KUKA KRL program: f1_Kuka_APT204T03S04.SRC

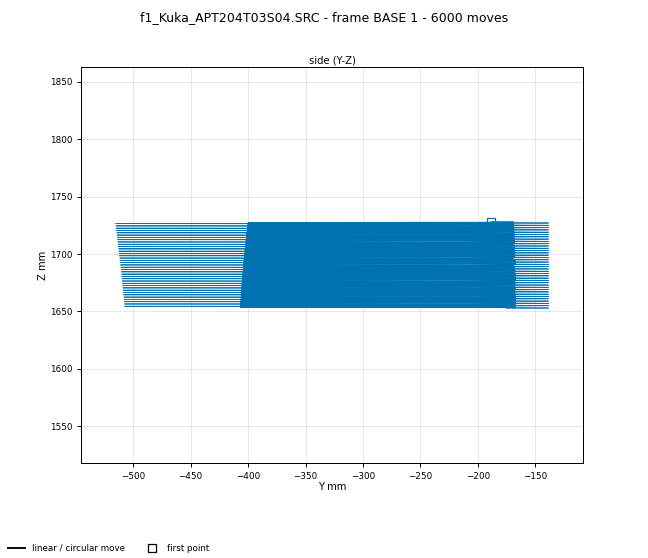
[picture p0: tool path of f1_Kuka_APT204T03S04.SRC in frame BASE 1, 6000 of 6001 moves have a stored position in this frame; points joined in program order, loops and branches not executed]
&ACCESS RVP
&REL 2
&PARAM TEMPLATE = C:\KRC\Roboter\Template\vorgabe
&PARAM EDITMASK = *
DEF f1_Kuka_APT204T03S04()


;FOLD INI;%{PE}%V3.2.0,%MKUKATPBASIS,%CINIT,%VCOMMON,%P
  ;FOLD BAS INI;%{E}%V3.2.0,%MKUKATPBASIS,%CINIT,%VINIT,%P
    GLOBAL INTERRUPT DECL 3 WHEN $STOPMESS==TRUE DO IR_STOPM ( )
    INTERRUPT ON 3
    BAS (#INITMOV,0 )
  ;ENDFOLD (BAS INI)
  ;FOLD USER INI;%{E}%V3.2.0,%MKUKATPUSER,%CINIT,%VINIT,%P
    ;Make your modifications here
  ;ENDFOLD (USER INI)
;ENDFOLD (INI)


;*** Make Null PTP Move
  PTP $pos_act

;*** Auto Load The Correct TOOL Data
  $tool=tool_data[3]

;*** Auto Load The Correct BASE Data
  $base=base_data[1]

  $ADVANCE = 5

;*** Restate Last Velocity
MMPM(30000.0)
SetRPM(6000)
LIN {X 0.021,Y -188.676,Z 1728.125,A 0.000,B 0.000,C 90.000,E1 22.408} C_DIS
LIN {X 0.032,Y -183.742,Z 1728.106,A 0.000,B 0.000,C 90.000,E1 19.087} C_DIS
LIN {X 0.032,Y -179.594,Z 1728.087,A 0.000,B 0.000,C 90.000,E1 15.733} C_DIS
LIN {X 0.087,Y -175.346,Z 1728.064,A 0.000,B 0.000,C 90.000,E1 11.478} C_DIS
LIN {X -0.024,Y -172.220,Z 1728.040,A 0.000,B 0.000,C 90.000,E1 7.239} C_DIS
LIN {X -0.008,Y -169.677,Z 1728.011,A 0.000,B 0.000,C 90.000,E1 2.064} C_DIS
LIN {X 0.036,Y -168.698,Z 1727.969,A 0.000,B 0.000,C 90.000,E1 354.318} C_DIS
LIN {X 0.059,Y -170.485,Z 1727.920,A 0.000,B 0.000,C 90.000,E1 345.644} C_DIS
LIN {X -0.021,Y -173.209,Z 1727.892,A 0.000,B 0.000,C 90.000,E1 340.496} C_DIS
LIN {X -0.074,Y -176.646,Z 1727.868,A 0.000,B 0.000,C 90.000,E1 336.230} C_DIS
LIN {X -0.056,Y -180.954,Z 1727.844,A 0.000,B 0.000,C 90.000,E1 331.975} C_DIS
LIN {X 0.018,Y -185.273,Z 1727.825,A 0.000,B 0.000,C 90.000,E1 328.584} C_DIS
LIN {X -0.017,Y -190.531,Z 1727.807,A 0.000,B 0.000,C 90.000,E1 325.261} C_DIS
LIN {X 0.064,Y -195.194,Z 1727.793,A 0.000,B 0.000,C 90.000,E1 322.763} C_DIS
LIN {X -0.077,Y -200.580,Z 1727.780,A 0.000,B 0.000,C 90.000,E1 320.356} C_DIS
LIN {X 0.012,Y -207.729,Z 1727.764,A 0.000,B 0.000,C 90.000,E1 317.514} C_DIS
LIN {X -0.032,Y -215.873,Z 1727.749,A 0.000,B 0.000,C 90.000,E1 314.757} C_DIS
LIN {X 0.037,Y -223.797,Z 1727.736,A 0.000,B 0.000,C 90.000,E1 312.405} C_DIS
LIN {X 0.016,Y -231.179,Z 1727.725,A 0.000,B 0.000,C 90.000,E1 310.496} C_DIS
LIN {X -0.046,Y -239.468,Z 1727.714,A 0.000,B 0.000,C 90.000,E1 308.624} C_DIS
LIN {X 0.070,Y -248.697,Z 1727.704,A 0.000,B 0.000,C 90.000,E1 306.744} C_DIS
LIN {X -0.140,Y -261.217,Z 1727.692,A 0.000,B 0.000,C 90.000,E1 304.612} C_DIS
LIN {X 0.044,Y -279.547,Z 1727.676,A 0.000,B 0.000,C 90.000,E1 301.750} C_DIS
LIN {X 0.044,Y -301.889,Z 1727.659,A 0.000,B 0.000,C 90.000,E1 298.693} C_DIS
LIN {X -0.011,Y -320.034,Z 1727.647,A 0.000,B 0.000,C 90.000,E1 296.411} C_DIS
LIN {X -0.057,Y -335.844,Z 1727.636,A 0.000,B 0.000,C 90.000,E1 294.515} C_DIS
LIN {X 0.099,Y -348.845,Z 1727.628,A 0.000,B 0.000,C 90.000,E1 292.950} C_DIS
LIN {X -0.069,Y -361.378,Z 1727.619,A 0.000,B 0.000,C 90.000,E1 291.461} C_DIS
LIN {X 0.072,Y -371.097,Z 1727.613,A 0.000,B 0.000,C 90.000,E1 290.248} C_DIS
LIN {X -0.125,Y -377.905,Z 1727.608,A 0.000,B 0.000,C 90.000,E1 289.396} C_DIS
LIN {X 0.102,Y -381.961,Z 1727.604,A 0.000,B 0.000,C 90.000,E1 288.779} C_DIS
LIN {X -0.113,Y -387.245,Z 1727.600,A 0.000,B 0.000,C 90.000,E1 287.946} C_DIS
LIN {X 0.057,Y -390.219,Z 1727.596,A 0.000,B 0.000,C 90.000,E1 287.347} C_DIS
LIN {X 0.030,Y -393.882,Z 1727.592,A 0.000,B 0.000,C 90.000,E1 286.496} C_DIS
LIN {X -0.134,Y -395.829,Z 1727.589,A 0.000,B 0.000,C 90.000,E1 285.953} C_DIS
LIN {X -0.018,Y -397.436,Z 1727.585,A 0.000,B 0.000,C 90.000,E1 285.371} C_DIS
LIN {X -0.169,Y -398.668,Z 1727.582,A 0.000,B 0.000,C 90.000,E1 284.828} C_DIS
LIN {X -0.025,Y -399.563,Z 1727.579,A 0.000,B 0.000,C 90.000,E1 284.245} C_DIS
LIN {X 0.225,Y -400.068,Z 1727.576,A 0.000,B 0.000,C 90.000,E1 283.647} C_DIS
LIN {X -0.004,Y -400.218,Z 1727.573,A 0.000,B 0.000,C 90.000,E1 283.119} C_DIS
LIN {X 0.160,Y -399.926,Z 1727.570,A 0.000,B 0.000,C 90.000,E1 282.535} C_DIS
LIN {X -0.063,Y -399.279,Z 1727.567,A 0.000,B 0.000,C 90.000,E1 282.007} C_DIS
LIN {X 0.103,Y -398.089,Z 1727.564,A 0.000,B 0.000,C 90.000,E1 281.422} C_DIS
LIN {X -0.126,Y -396.417,Z 1727.560,A 0.000,B 0.000,C 90.000,E1 280.894} C_DIS
LIN {X 0.026,Y -394.202,Z 1727.557,A 0.000,B 0.000,C 90.000,E1 280.310} C_DIS
LIN {X 0.159,Y -391.354,Z 1727.554,A 0.000,B 0.000,C 90.000,E1 279.726} C_DIS
LIN {X -0.031,Y -379.747,Z 1727.543,A 0.000,B 0.000,C 90.000,E1 277.757} C_DIS
LIN {X -0.040,Y -376.170,Z 1727.540,A 0.000,B 0.000,C 90.000,E1 277.182} C_DIS
LIN {X -0.068,Y -372.156,Z 1727.537,A 0.000,B 0.000,C 90.000,E1 276.606} C_DIS
LIN {X -0.115,Y -367.505,Z 1727.533,A 0.000,B 0.000,C 90.000,E1 276.030} C_DIS
LIN {X -0.141,Y -362.126,Z 1727.530,A 0.000,B 0.000,C 90.000,E1 275.448} C_DIS
LIN {X -0.100,Y -356.268,Z 1727.527,A 0.000,B 0.000,C 90.000,E1 274.878} C_DIS
LIN {X -0.130,Y -350.292,Z 1727.524,A 0.000,B 0.000,C 90.000,E1 274.359} C_DIS
LIN {X 0.065,Y -344.121,Z 1727.521,A 0.000,B 0.000,C 90.000,E1 273.841} C_DIS
LIN {X 0.135,Y -337.795,Z 1727.519,A 0.000,B 0.000,C 90.000,E1 273.383} C_DIS
LIN {X 0.110,Y -331.427,Z 1727.517,A 0.000,B 0.000,C 90.000,E1 272.980} C_DIS
LIN {X -0.017,Y -321.523,Z 1727.514,A 0.000,B 0.000,C 90.000,E1 272.465} C_DIS
LIN {X -0.159,Y -314.709,Z 1727.512,A 0.000,B 0.000,C 90.000,E1 272.178} C_DIS
LIN {X -0.109,Y -307.490,Z 1727.510,A 0.000,B 0.000,C 90.000,E1 271.892} C_DIS
LIN {X -0.010,Y -296.875,Z 1727.509,A 0.000,B 0.000,C 90.000,E1 271.547} C_DIS
LIN {X -0.063,Y -289.643,Z 1727.508,A 0.000,B 0.000,C 90.000,E1 271.375} C_DIS
LIN {X -0.035,Y -277.079,Z 1727.506,A 0.000,B 0.000,C 90.000,E1 271.146} C_DIS
LIN {X -0.052,Y -264.431,Z 1727.505,A 0.000,B 0.000,C 90.000,E1 270.974} C_DIS
LIN {X -0.027,Y -253.912,Z 1727.505,A 0.000,B 0.000,C 90.000,E1 270.859} C_DIS
LIN {X -0.046,Y -239.564,Z 1727.504,A 0.000,B 0.000,C 90.000,E1 270.802} C_DIS
LIN {X -0.067,Y -181.507,Z 1727.504,A 0.000,B 0.000,C 90.000,E1 270.802} C_DIS
LIN {X -0.020,Y -181.537,Z 1727.499,A 0.000,B 0.000,C 90.000,E1 269.885} C_DIS
LIN {X -0.036,Y -180.813,Z 1727.471,A 0.000,B 0.000,C 90.000,E1 264.837} C_DIS
LIN {X 0.041,Y -178.916,Z 1727.443,A 0.000,B 0.000,C 90.000,E1 259.746} C_DIS
LIN {X -0.050,Y -175.961,Z 1727.415,A 0.000,B 0.000,C 90.000,E1 254.685} C_DIS
LIN {X 0.067,Y -175.435,Z 1727.410,A 0.000,B 0.000,C 90.000,E1 253.795} C_DIS
LIN {X 0.069,Y -172.193,Z 1727.386,A 0.000,B 0.000,C 90.000,E1 249.518} C_DIS
LIN {X 0.046,Y -171.666,Z 1727.382,A 0.000,B 0.000,C 90.000,E1 248.666} C_DIS
LIN {X 0.029,Y -167.891,Z 1727.358,A 0.000,B 0.000,C 90.000,E1 244.357} C_DIS
LIN {X 0.045,Y -166.629,Z 1727.348,A 0.000,B 0.000,C 90.000,E1 242.615} C_DIS
LIN {X 0.037,Y -162.615,Z 1727.324,A 0.000,B 0.000,C 90.000,E1 238.250} C_DIS
LIN {X 0.012,Y -161.301,Z 1727.314,A 0.000,B 0.000,C 90.000,E1 236.501} C_DIS
LIN {X 0.045,Y -157.299,Z 1727.289,A 0.000,B 0.000,C 90.000,E1 232.065} C_DIS
LIN {X 0.074,Y -155.274,Z 1727.275,A 0.000,B 0.000,C 90.000,E1 229.380} C_DIS
LIN {X 0.002,Y -151.641,Z 1727.250,A 0.000,B 0.000,C 90.000,E1 224.919} C_DIS
LIN {X 0.049,Y -150.509,Z 1727.240,A 0.000,B 0.000,C 90.000,E1 223.095} C_DIS
LIN {X -0.037,Y -147.234,Z 1727.214,A 0.000,B 0.000,C 90.000,E1 218.588} C_DIS
LIN {X 0.048,Y -145.257,Z 1727.194,A 0.000,B 0.000,C 90.000,E1 214.898} C_DIS
LIN {X -0.036,Y -142.370,Z 1727.163,A 0.000,B 0.000,C 90.000,E1 209.411} C_DIS
LIN {X 0.085,Y -141.755,Z 1727.153,A 0.000,B 0.000,C 90.000,E1 207.513} C_DIS
LIN {X 0.010,Y -139.497,Z 1727.117,A 0.000,B 0.000,C 90.000,E1 201.046} C_DIS
LIN {X 0.047,Y -139.002,Z 1727.101,A 0.000,B 0.000,C 90.000,E1 198.236} C_DIS
LIN {X 0.003,Y -138.338,Z 1727.055,A 0.000,B 0.000,C 90.000,E1 189.849} C_DIS
LIN {X 0.025,Y -139.408,Z 1727.008,A 0.000,B 0.000,C 90.000,E1 181.432} C_DIS
LIN {X -0.062,Y -141.318,Z 1726.972,A 0.000,B 0.000,C 90.000,E1 174.951} C_DIS
LIN {X 0.037,Y -142.677,Z 1726.956,A 0.000,B 0.000,C 90.000,E1 172.129} C_DIS
LIN {X 0.017,Y -145.032,Z 1726.931,A 0.000,B 0.000,C 90.000,E1 167.521} C_DIS
LIN {X -0.026,Y -147.657,Z 1726.910,A 0.000,B 0.000,C 90.000,E1 163.866} C_DIS
LIN {X 0.050,Y -150.295,Z 1726.890,A 0.000,B 0.000,C 90.000,E1 160.188} C_DIS
LIN {X -0.079,Y -153.704,Z 1726.870,A 0.000,B 0.000,C 90.000,E1 156.613} C_DIS
LIN {X -0.024,Y -157.118,Z 1726.850,A 0.000,B 0.000,C 90.000,E1 152.999} C_DIS
LIN {X 0.052,Y -161.260,Z 1726.830,A 0.000,B 0.000,C 90.000,E1 149.410} C_DIS
LIN {X -0.020,Y -164.379,Z 1726.815,A 0.000,B 0.000,C 90.000,E1 146.786} C_DIS
LIN {X -0.033,Y -169.054,Z 1726.796,A 0.000,B 0.000,C 90.000,E1 143.290} C_DIS
LIN {X 0.019,Y -171.615,Z 1726.786,A 0.000,B 0.000,C 90.000,E1 141.537} C_DIS
LIN {X 0.067,Y -176.571,Z 1726.767,A 0.000,B 0.000,C 90.000,E1 138.081} C_DIS
LIN {X -0.060,Y -180.869,Z 1726.753,A 0.000,B 0.000,C 90.000,E1 135.567} C_DIS
LIN {X 0.062,Y -186.283,Z 1726.734,A 0.000,B 0.000,C 90.000,E1 132.162} C_DIS
LIN {X -0.017,Y -190.918,Z 1726.720,A 0.000,B 0.000,C 90.000,E1 129.688} C_DIS
LIN {X 0.051,Y -196.685,Z 1726.702,A 0.000,B 0.000,C 90.000,E1 126.377} C_DIS
LIN {X 0.081,Y -199.929,Z 1726.693,A 0.000,B 0.000,C 90.000,E1 124.739} C_DIS
LIN {X -0.026,Y -205.846,Z 1726.675,A 0.000,B 0.000,C 90.000,E1 121.544} C_DIS
LIN {X -0.035,Y -209.790,Z 1726.664,A 0.000,B 0.000,C 90.000,E1 119.617} C_DIS
LIN {X -0.091,Y -333.994,Z 1726.664,A 0.000,B 0.000,C 90.000,E1 119.617} C_DIS
LIN {X -0.010,Y -338.536,Z 1726.664,A 0.000,B 0.000,C 90.000,E1 119.489} C_DIS
LIN {X 0.072,Y -340.616,Z 1726.663,A 0.000,B 0.000,C 90.000,E1 119.361} C_DIS
LIN {X -0.059,Y -343.462,Z 1726.662,A 0.000,B 0.000,C 90.000,E1 119.155} C_DIS
LIN {X -0.065,Y -347.189,Z 1726.659,A 0.000,B 0.000,C 90.000,E1 118.693} C_DIS
LIN {X 0.099,Y -348.907,Z 1726.658,A 0.000,B 0.000,C 90.000,E1 118.359} C_DIS
LIN {X -0.093,Y -361.834,Z 1726.643,A 0.000,B 0.000,C 90.000,E1 115.668} C_DIS
LIN {X -0.076,Y -376.245,Z 1726.628,A 0.000,B 0.000,C 90.000,E1 113.003} C_DIS
LIN {X 0.097,Y -390.434,Z 1726.615,A 0.000,B 0.000,C 90.000,E1 110.663} C_DIS
LIN {X -0.010,Y -406.020,Z 1726.602,A 0.000,B 0.000,C 90.000,E1 108.417} C_DIS
LIN {X 0.018,Y -423.110,Z 1726.590,A 0.000,B 0.000,C 90.000,E1 106.205} C_DIS
LIN {X -0.058,Y -441.822,Z 1726.578,A 0.000,B 0.000,C 90.000,E1 104.064} C_DIS
LIN {X 0.100,Y -461.716,Z 1726.567,A 0.000,B 0.000,C 90.000,E1 102.007} C_DIS
LIN {X 0.139,Y -484.774,Z 1726.555,A 0.000,B 0.000,C 90.000,E1 99.905} C_DIS
LIN {X 0.179,Y -508.285,Z 1726.545,A 0.000,B 0.000,C 90.000,E1 97.992} C_DIS
LIN {X -0.039,Y -510.226,Z 1726.543,A 0.000,B 0.000,C 90.000,E1 97.814} C_DIS
LIN {X -0.158,Y -511.971,Z 1726.542,A 0.000,B 0.000,C 90.000,E1 97.587} C_DIS
LIN {X -0.211,Y -513.277,Z 1726.541,A 0.000,B 0.000,C 90.000,E1 97.352} C_DIS
LIN {X 0.150,Y -514.880,Z 1726.538,A 0.000,B 0.000,C 90.000,E1 96.834} C_DIS
LIN {X 0.006,Y -515.381,Z 1726.535,A 0.000,B 0.000,C 90.000,E1 96.372} C_DIS
LIN {X -0.129,Y -514.864,Z 1726.533,A 0.000,B 0.000,C 90.000,E1 95.910} C_DIS
LIN {X 0.249,Y -513.239,Z 1726.530,A 0.000,B 0.000,C 90.000,E1 95.391} C_DIS
LIN {X 0.157,Y -511.916,Z 1726.529,A 0.000,B 0.000,C 90.000,E1 95.163} C_DIS
LIN {X 0.131,Y -501.107,Z 1726.521,A 0.000,B 0.000,C 90.000,E1 93.726} C_DIS
LIN {X -0.234,Y -488.498,Z 1726.511,A 0.000,B 0.000,C 90.000,E1 92.064} C_DIS
LIN {X 0.126,Y -475.702,Z 1726.502,A 0.000,B 0.000,C 90.000,E1 90.286} C_DIS
LIN {X -0.052,Y -464.718,Z 1726.493,A 0.000,B 0.000,C 90.000,E1 88.797} C_DIS
LIN {X -0.170,Y -451.882,Z 1726.483,A 0.000,B 0.000,C 90.000,E1 87.020} C_DIS
LIN {X 0.127,Y -437.184,Z 1726.472,A 0.000,B 0.000,C 90.000,E1 84.894} C_DIS
LIN {X -0.047,Y -424.340,Z 1726.461,A 0.000,B 0.000,C 90.000,E1 83.053} C_DIS
LIN {X -0.059,Y -406.525,Z 1726.446,A 0.000,B 0.000,C 90.000,E1 80.330} C_DIS
LIN {X 0.031,Y -389.797,Z 1726.431,A 0.000,B 0.000,C 90.000,E1 77.521} C_DIS
LIN {X 0.060,Y -377.038,Z 1726.418,A 0.000,B 0.000,C 90.000,E1 75.227} C_DIS
LIN {X -0.004,Y -366.137,Z 1726.407,A 0.000,B 0.000,C 90.000,E1 73.196} C_DIS
LIN {X 0.137,Y -352.444,Z 1726.392,A 0.000,B 0.000,C 90.000,E1 70.496} C_DIS
LIN {X -0.072,Y -339.450,Z 1726.377,A 0.000,B 0.000,C 90.000,E1 67.794} C_DIS
LIN {X -0.006,Y -329.467,Z 1726.365,A 0.000,B 0.000,C 90.000,E1 65.613} C_DIS
LIN {X 0.136,Y -317.003,Z 1726.349,A 0.000,B 0.000,C 90.000,E1 62.743} C_DIS
LIN {X 0.005,Y -307.384,Z 1726.336,A 0.000,B 0.000,C 90.000,E1 60.511} C_DIS
LIN {X 0.090,Y -297.798,Z 1726.323,A 0.000,B 0.000,C 90.000,E1 58.201} C_DIS
LIN {X 0.015,Y -288.121,Z 1726.310,A 0.000,B 0.000,C 90.000,E1 55.881} C_DIS
LIN {X 0.057,Y -278.348,Z 1726.297,A 0.000,B 0.000,C 90.000,E1 53.497} C_DIS
LIN {X -0.007,Y -268.542,Z 1726.284,A 0.000,B 0.000,C 90.000,E1 51.090} C_DIS
LIN {X 0.107,Y -257.502,Z 1726.268,A 0.000,B 0.000,C 90.000,E1 48.243} C_DIS
LIN {X 0.086,Y -245.401,Z 1726.250,A 0.000,B 0.000,C 90.000,E1 45.000} C_DIS
LIN {X 0.076,Y -234.032,Z 1726.232,A 0.000,B 0.000,C 90.000,E1 41.676} C_DIS
LIN {X 0.026,Y -224.586,Z 1726.215,A 0.000,B 0.000,C 90.000,E1 38.669} C_DIS
LIN {X -0.089,Y -217.046,Z 1726.200,A 0.000,B 0.000,C 90.000,E1 36.011} C_DIS
LIN {X -0.046,Y -209.230,Z 1726.183,A 0.000,B 0.000,C 90.000,E1 32.880} C_DIS
LIN {X 0.102,Y -202.113,Z 1726.165,A 0.000,B 0.000,C 90.000,E1 29.667} C_DIS
LIN {X -0.046,Y -195.705,Z 1726.147,A 0.000,B 0.000,C 90.000,E1 26.488} C_DIS
LIN {X 0.008,Y -189.907,Z 1726.129,A 0.000,B 0.000,C 90.000,E1 23.206} C_DIS
LIN {X -0.020,Y -185.956,Z 1726.115,A 0.000,B 0.000,C 90.000,E1 20.737} C_DIS
LIN {X -0.027,Y -181.437,Z 1726.097,A 0.000,B 0.000,C 90.000,E1 17.402} C_DIS
LIN {X -0.002,Y -176.803,Z 1726.073,A 0.000,B 0.000,C 90.000,E1 13.175} C_DIS
LIN {X -0.012,Y -173.238,Z 1726.050,A 0.000,B 0.000,C 90.000,E1 8.916} C_DIS
LIN {X 0.080,Y -170.204,Z 1726.021,A 0.000,B 0.000,C 90.000,E1 3.726} C_DIS
LIN {X 0.031,Y -168.549,Z 1725.969,A 0.000,B 0.000,C 90.000,E1 354.318} C_DIS
LIN {X 0.047,Y -170.375,Z 1725.920,A 0.000,B 0.000,C 90.000,E1 345.644} C_DIS
LIN {X -0.036,Y -173.138,Z 1725.892,A 0.000,B 0.000,C 90.000,E1 340.496} C_DIS
LIN {X 0.069,Y -176.589,Z 1725.868,A 0.000,B 0.000,C 90.000,E1 336.177} C_DIS
LIN {X -0.077,Y -180.926,Z 1725.844,A 0.000,B 0.000,C 90.000,E1 331.975} C_DIS
LIN {X -0.004,Y -185.262,Z 1725.825,A 0.000,B 0.000,C 90.000,E1 328.584} C_DIS
LIN {X -0.040,Y -190.547,Z 1725.807,A 0.000,B 0.000,C 90.000,E1 325.261} C_DIS
LIN {X 0.041,Y -195.244,Z 1725.793,A 0.000,B 0.000,C 90.000,E1 322.763} C_DIS
LIN {X 0.050,Y -201.625,Z 1725.777,A 0.000,B 0.000,C 90.000,E1 319.908} C_DIS
LIN {X 0.031,Y -208.936,Z 1725.762,A 0.000,B 0.000,C 90.000,E1 317.106} C_DIS
LIN {X 0.008,Y -217.290,Z 1725.746,A 0.000,B 0.000,C 90.000,E1 314.352} C_DIS
LIN {X 0.105,Y -225.385,Z 1725.734,A 0.000,B 0.000,C 90.000,E1 312.000} C_DIS
LIN {X 0.104,Y -232.950,Z 1725.723,A 0.000,B 0.000,C 90.000,E1 310.092} C_DIS
LIN {X -0.076,Y -241.392,Z 1725.712,A 0.000,B 0.000,C 90.000,E1 308.257} C_DIS
LIN {X 0.065,Y -250.866,Z 1725.702,A 0.000,B 0.000,C 90.000,E1 306.377} C_DIS
LIN {X 0.109,Y -263.640,Z 1725.690,A 0.000,B 0.000,C 90.000,E1 304.199} C_DIS
LIN {X -0.011,Y -282.177,Z 1725.675,A 0.000,B 0.000,C 90.000,E1 301.416} C_DIS
LIN {X 0.056,Y -302.095,Z 1725.659,A 0.000,B 0.000,C 90.000,E1 298.693} C_DIS
LIN {X 0.005,Y -320.201,Z 1725.647,A 0.000,B 0.000,C 90.000,E1 296.411} C_DIS
LIN {X -0.055,Y -335.995,Z 1725.636,A 0.000,B 0.000,C 90.000,E1 294.515} C_DIS
LIN {X 0.102,Y -348.973,Z 1725.628,A 0.000,B 0.000,C 90.000,E1 292.950} C_DIS
LIN {X -0.065,Y -361.513,Z 1725.619,A 0.000,B 0.000,C 90.000,E1 291.461} C_DIS
LIN {X 0.078,Y -371.239,Z 1725.613,A 0.000,B 0.000,C 90.000,E1 290.248} C_DIS
LIN {X -0.117,Y -378.062,Z 1725.608,A 0.000,B 0.000,C 90.000,E1 289.396} C_DIS
LIN {X 0.112,Y -382.108,Z 1725.604,A 0.000,B 0.000,C 90.000,E1 288.779} C_DIS
LIN {X -0.103,Y -387.404,Z 1725.600,A 0.000,B 0.000,C 90.000,E1 287.946} C_DIS
LIN {X 0.068,Y -390.382,Z 1725.596,A 0.000,B 0.000,C 90.000,E1 287.347} C_DIS
LIN {X 0.043,Y -394.065,Z 1725.592,A 0.000,B 0.000,C 90.000,E1 286.496} C_DIS
LIN {X -0.120,Y -396.048,Z 1725.589,A 0.000,B 0.000,C 90.000,E1 285.953} C_DIS
LIN {X -0.003,Y -397.675,Z 1725.585,A 0.000,B 0.000,C 90.000,E1 285.371} C_DIS
LIN {X -0.152,Y -398.895,Z 1725.582,A 0.000,B 0.000,C 90.000,E1 284.828} C_DIS
LIN {X -0.007,Y -399.799,Z 1725.579,A 0.000,B 0.000,C 90.000,E1 284.245} C_DIS
LIN {X -0.144,Y -400.296,Z 1725.576,A 0.000,B 0.000,C 90.000,E1 283.703} C_DIS
LIN {X 0.017,Y -400.428,Z 1725.573,A 0.000,B 0.000,C 90.000,E1 283.119} C_DIS
LIN {X 0.183,Y -400.155,Z 1725.570,A 0.000,B 0.000,C 90.000,E1 282.535} C_DIS
LIN {X -0.040,Y -399.488,Z 1725.567,A 0.000,B 0.000,C 90.000,E1 282.007} C_DIS
LIN {X 0.128,Y -398.290,Z 1725.564,A 0.000,B 0.000,C 90.000,E1 281.422} C_DIS
LIN {X -0.100,Y -396.610,Z 1725.560,A 0.000,B 0.000,C 90.000,E1 280.894} C_DIS
LIN {X 0.052,Y -394.381,Z 1725.557,A 0.000,B 0.000,C 90.000,E1 280.310} C_DIS
LIN {X 0.186,Y -391.546,Z 1725.554,A 0.000,B 0.000,C 90.000,E1 279.726} C_DIS
LIN {X 0.000,Y -379.916,Z 1725.543,A 0.000,B 0.000,C 90.000,E1 277.757} C_DIS
LIN {X 0.006,Y -374.386,Z 1725.538,A 0.000,B 0.000,C 90.000,E1 276.891} C_DIS
LIN {X -0.033,Y -370.048,Z 1725.535,A 0.000,B 0.000,C 90.000,E1 276.315} C_DIS
LIN {X -0.093,Y -364.999,Z 1725.532,A 0.000,B 0.000,C 90.000,E1 275.739} C_DIS
LIN {X 0.179,Y -359.290,Z 1725.529,A 0.000,B 0.000,C 90.000,E1 275.106} C_DIS
LIN {X 0.013,Y -353.325,Z 1725.526,A 0.000,B 0.000,C 90.000,E1 274.588} C_DIS
LIN {X 0.089,Y -347.232,Z 1725.523,A 0.000,B 0.000,C 90.000,E1 274.073} C_DIS
LIN {X 0.076,Y -340.957,Z 1725.520,A 0.000,B 0.000,C 90.000,E1 273.612} C_DIS
LIN {X -0.061,Y -334.532,Z 1725.518,A 0.000,B 0.000,C 90.000,E1 273.212} C_DIS
LIN {X 0.026,Y -327.904,Z 1725.516,A 0.000,B 0.000,C 90.000,E1 272.808} C_DIS
LIN {X 0.012,Y -321.289,Z 1725.514,A 0.000,B 0.000,C 90.000,E1 272.465} C_DIS
LIN {X -0.146,Y -314.295,Z 1725.512,A 0.000,B 0.000,C 90.000,E1 272.178} C_DIS
LIN {X -0.009,Y -303.873,Z 1725.510,A 0.000,B 0.000,C 90.000,E1 271.776} C_DIS
LIN {X -0.087,Y -293.320,Z 1725.508,A 0.000,B 0.000,C 90.000,E1 271.489} C_DIS
LIN {X -0.080,Y -285.623,Z 1725.507,A 0.000,B 0.000,C 90.000,E1 271.318} C_DIS
LIN {X 0.077,Y -269.385,Z 1725.506,A 0.000,B 0.000,C 90.000,E1 271.031} C_DIS
LIN {X 0.089,Y -255.161,Z 1725.505,A 0.000,B 0.000,C 90.000,E1 270.859} C_DIS
LIN {X 0.059,Y -239.893,Z 1725.505,A 0.000,B 0.000,C 90.000,E1 270.802} C_DIS
LIN {X 0.014,Y -181.500,Z 1725.505,A 0.000,B 0.000,C 90.000,E1 270.802} C_DIS
LIN {X 0.068,Y -181.543,Z 1725.500,A 0.000,B 0.000,C 90.000,E1 269.885} C_DIS
LIN {X 0.052,Y -180.822,Z 1725.471,A 0.000,B 0.000,C 90.000,E1 264.837} C_DIS
LIN {X -0.048,Y -178.926,Z 1725.443,A 0.000,B 0.000,C 90.000,E1 259.803} C_DIS
LIN {X -0.010,Y -175.973,Z 1725.415,A 0.000,B 0.000,C 90.000,E1 254.700} C_DIS
LIN {X -0.065,Y -175.459,Z 1725.410,A 0.000,B 0.000,C 90.000,E1 253.866} C_DIS
LIN {X -0.007,Y -172.210,Z 1725.386,A 0.000,B 0.000,C 90.000,E1 249.571} C_DIS
LIN {X -0.029,Y -171.686,Z 1725.382,A 0.000,B 0.000,C 90.000,E1 248.720} C_DIS
LIN {X -0.039,Y -167.912,Z 1725.358,A 0.000,B 0.000,C 90.000,E1 244.409} C_DIS
LIN {X -0.020,Y -166.654,Z 1725.348,A 0.000,B 0.000,C 90.000,E1 242.666} C_DIS
LIN {X 0.034,Y -162.638,Z 1725.324,A 0.000,B 0.000,C 90.000,E1 238.280} C_DIS
LIN {X -0.041,Y -161.325,Z 1725.314,A 0.000,B 0.000,C 90.000,E1 236.548} C_DIS
LIN {X 0.002,Y -157.321,Z 1725.290,A 0.000,B 0.000,C 90.000,E1 232.110} C_DIS
LIN {X -0.065,Y -155.301,Z 1725.275,A 0.000,B 0.000,C 90.000,E1 229.461} C_DIS
LIN {X 0.081,Y -151.661,Z 1725.250,A 0.000,B 0.000,C 90.000,E1 224.919} C_DIS
LIN {X 0.018,Y -150.527,Z 1725.240,A 0.000,B 0.000,C 90.000,E1 223.137} C_DIS
LIN {X -0.051,Y -147.252,Z 1725.214,A 0.000,B 0.000,C 90.000,E1 218.624} C_DIS
LIN {X 0.005,Y -145.277,Z 1725.194,A 0.000,B 0.000,C 90.000,E1 214.945} C_DIS
LIN {X 0.039,Y -142.381,Z 1725.163,A 0.000,B 0.000,C 90.000,E1 209.411} C_DIS
LIN {X -0.039,Y -141.359,Z 1725.148,A 0.000,B 0.000,C 90.000,E1 206.668} C_DIS
LIN {X 0.071,Y -139.342,Z 1725.112,A 0.000,B 0.000,C 90.000,E1 200.120} C_DIS
LIN {X -0.011,Y -139.010,Z 1725.102,A 0.000,B 0.000,C 90.000,E1 198.290} C_DIS
LIN {X -0.059,Y -138.341,Z 1725.055,A 0.000,B 0.000,C 90.000,E1 189.905} C_DIS
LIN {X -0.039,Y -139.400,Z 1725.008,A 0.000,B 0.000,C 90.000,E1 181.489} C_DIS
LIN {X 0.014,Y -141.304,Z 1724.972,A 0.000,B 0.000,C 90.000,E1 174.951} C_DIS
LIN {X -0.028,Y -142.665,Z 1724.957,A 0.000,B 0.000,C 90.000,E1 172.186} C_DIS
LIN {X -0.079,Y -145.012,Z 1724.931,A 0.000,B 0.000,C 90.000,E1 167.589} C_DIS
LIN {X 0.052,Y -147.639,Z 1724.911,A 0.000,B 0.000,C 90.000,E1 163.866} C_DIS
LIN {X -0.012,Y -150.271,Z 1724.890,A 0.000,B 0.000,C 90.000,E1 160.242} C_DIS
LIN {X 0.001,Y -153.672,Z 1724.870,A 0.000,B 0.000,C 90.000,E1 156.613} C_DIS
LIN {X 0.057,Y -157.087,Z 1724.850,A 0.000,B 0.000,C 90.000,E1 152.999} C_DIS
LIN {X -0.004,Y -161.222,Z 1724.830,A 0.000,B 0.000,C 90.000,E1 149.459} C_DIS
LIN {X 0.080,Y -163.312,Z 1724.820,A 0.000,B 0.000,C 90.000,E1 147.661} C_DIS
LIN {X -0.048,Y -167.761,Z 1724.801,A 0.000,B 0.000,C 90.000,E1 144.196} C_DIS
LIN {X 0.104,Y -171.578,Z 1724.786,A 0.000,B 0.000,C 90.000,E1 141.537} C_DIS
LIN {X -0.096,Y -176.527,Z 1724.767,A 0.000,B 0.000,C 90.000,E1 138.162} C_DIS
LIN {X 0.028,Y -180.825,Z 1724.753,A 0.000,B 0.000,C 90.000,E1 135.567} C_DIS
LIN {X 0.013,Y -186.235,Z 1724.734,A 0.000,B 0.000,C 90.000,E1 132.204} C_DIS
LIN {X -0.048,Y -190.871,Z 1724.721,A 0.000,B 0.000,C 90.000,E1 129.725} C_DIS
LIN {X -0.015,Y -196.634,Z 1724.702,A 0.000,B 0.000,C 90.000,E1 126.423} C_DIS
LIN {X -0.103,Y -199.873,Z 1724.693,A 0.000,B 0.000,C 90.000,E1 124.818} C_DIS
LIN {X 0.093,Y -204.269,Z 1724.680,A 0.000,B 0.000,C 90.000,E1 122.339} C_DIS
LIN {X 0.061,Y -209.734,Z 1724.665,A 0.000,B 0.000,C 90.000,E1 119.617} C_DIS
LIN {X 0.061,Y -334.184,Z 1724.665,A 0.000,B 0.000,C 90.000,E1 119.617} C_DIS
LIN {X -0.151,Y -338.440,Z 1724.664,A 0.000,B 0.000,C 90.000,E1 119.539} C_DIS
LIN {X -0.069,Y -340.506,Z 1724.663,A 0.000,B 0.000,C 90.000,E1 119.411} C_DIS
LIN {X 0.097,Y -343.339,Z 1724.662,A 0.000,B 0.000,C 90.000,E1 119.155} C_DIS
LIN {X 0.084,Y -347.067,Z 1724.659,A 0.000,B 0.000,C 90.000,E1 118.693} C_DIS
LIN {X -0.058,Y -348.777,Z 1724.658,A 0.000,B 0.000,C 90.000,E1 118.409} C_DIS
LIN {X 0.058,Y -361.691,Z 1724.643,A 0.000,B 0.000,C 90.000,E1 115.668} C_DIS
LIN {X -0.070,Y -376.087,Z 1724.628,A 0.000,B 0.000,C 90.000,E1 113.025} C_DIS
LIN {X 0.113,Y -390.262,Z 1724.615,A 0.000,B 0.000,C 90.000,E1 110.684} C_DIS
LIN {X 0.147,Y -405.833,Z 1724.602,A 0.000,B 0.000,C 90.000,E1 108.417} C_DIS
LIN {X 0.176,Y -422.907,Z 1724.590,A 0.000,B 0.000,C 90.000,E1 106.205} C_DIS
LIN {X 0.102,Y -441.603,Z 1724.578,A 0.000,B 0.000,C 90.000,E1 104.064} C_DIS
LIN {X -0.197,Y -461.489,Z 1724.567,A 0.000,B 0.000,C 90.000,E1 102.063} C_DIS
LIN {X -0.192,Y -484.541,Z 1724.555,A 0.000,B 0.000,C 90.000,E1 99.962} C_DIS
LIN {X -0.185,Y -508.048,Z 1724.545,A 0.000,B 0.000,C 90.000,E1 98.049} C_DIS
LIN {X 0.099,Y -509.989,Z 1724.543,A 0.000,B 0.000,C 90.000,E1 97.814} C_DIS
LIN {X -0.020,Y -511.734,Z 1724.542,A 0.000,B 0.000,C 90.000,E1 97.587} C_DIS
LIN {X -0.072,Y -513.038,Z 1724.541,A 0.000,B 0.000,C 90.000,E1 97.352} C_DIS
LIN {X -0.224,Y -514.635,Z 1724.538,A 0.000,B 0.000,C 90.000,E1 96.891} C_DIS
LIN {X 0.142,Y -515.135,Z 1724.536,A 0.000,B 0.000,C 90.000,E1 96.372} C_DIS
LIN {X 0.005,Y -514.617,Z 1724.533,A 0.000,B 0.000,C 90.000,E1 95.910} C_DIS
LIN {X -0.129,Y -512.990,Z 1724.530,A 0.000,B 0.000,C 90.000,E1 95.448} C_DIS
LIN {X -0.221,Y -511.668,Z 1724.529,A 0.000,B 0.000,C 90.000,E1 95.220} C_DIS
LIN {X -0.130,Y -502.681,Z 1724.522,A 0.000,B 0.000,C 90.000,E1 94.012} C_DIS
LIN {X 0.020,Y -490.069,Z 1724.513,A 0.000,B 0.000,C 90.000,E1 92.293} C_DIS
LIN {X 0.096,Y -479.126,Z 1724.505,A 0.000,B 0.000,C 90.000,E1 90.802} C_DIS
LIN {X -0.214,Y -466.337,Z 1724.495,A 0.000,B 0.000,C 90.000,E1 89.083} C_DIS
LIN {X -0.075,Y -451.649,Z 1724.483,A 0.000,B 0.000,C 90.000,E1 87.020} C_DIS
LIN {X 0.214,Y -436.922,Z 1724.472,A 0.000,B 0.000,C 90.000,E1 84.894} C_DIS
LIN {X 0.032,Y -424.062,Z 1724.461,A 0.000,B 0.000,C 90.000,E1 83.053} C_DIS
LIN {X 0.009,Y -406.241,Z 1724.446,A 0.000,B 0.000,C 90.000,E1 80.330} C_DIS
LIN {X 0.088,Y -389.491,Z 1724.431,A 0.000,B 0.000,C 90.000,E1 77.521} C_DIS
LIN {X 0.107,Y -376.706,Z 1724.418,A 0.000,B 0.000,C 90.000,E1 75.227} C_DIS
LIN {X 0.035,Y -365.798,Z 1724.407,A 0.000,B 0.000,C 90.000,E1 73.196} C_DIS
LIN {X -0.167,Y -352.080,Z 1724.392,A 0.000,B 0.000,C 90.000,E1 70.550} C_DIS
LIN {X -0.054,Y -339.064,Z 1724.377,A 0.000,B 0.000,C 90.000,E1 67.794} C_DIS
LIN {X 0.003,Y -329.044,Z 1724.365,A 0.000,B 0.000,C 90.000,E1 65.613} C_DIS
LIN {X 0.133,Y -316.569,Z 1724.349,A 0.000,B 0.000,C 90.000,E1 62.743} C_DIS
LIN {X -0.054,Y -308.337,Z 1724.338,A 0.000,B 0.000,C 90.000,E1 60.845} C_DIS
LIN {X 0.070,Y -297.413,Z 1724.323,A 0.000,B 0.000,C 90.000,E1 58.201} C_DIS
LIN {X 0.003,Y -289.130,Z 1724.312,A 0.000,B 0.000,C 90.000,E1 56.215} C_DIS
LIN {X 0.067,Y -279.379,Z 1724.299,A 0.000,B 0.000,C 90.000,E1 53.829} C_DIS
LIN {X -0.132,Y -269.564,Z 1724.286,A 0.000,B 0.000,C 90.000,E1 51.457} C_DIS
LIN {X 0.015,Y -258.519,Z 1724.270,A 0.000,B 0.000,C 90.000,E1 48.609} C_DIS
LIN {X 0.031,Y -246.336,Z 1724.252,A 0.000,B 0.000,C 90.000,E1 45.364} C_DIS
LIN {X 0.045,Y -234.899,Z 1724.234,A 0.000,B 0.000,C 90.000,E1 42.043} C_DIS
LIN {X 0.014,Y -225.387,Z 1724.217,A 0.000,B 0.000,C 90.000,E1 39.036} C_DIS
LIN {X 0.020,Y -216.779,Z 1724.200,A 0.000,B 0.000,C 90.000,E1 35.964} C_DIS
LIN {X 0.059,Y -208.994,Z 1724.182,A 0.000,B 0.000,C 90.000,E1 32.832} C_DIS
LIN {X 0.028,Y -201.941,Z 1724.165,A 0.000,B 0.000,C 90.000,E1 29.667} C_DIS
LIN {X 0.053,Y -195.553,Z 1724.147,A 0.000,B 0.000,C 90.000,E1 26.437} C_DIS
LIN {X 0.094,Y -188.395,Z 1724.124,A 0.000,B 0.000,C 90.000,E1 22.333} C_DIS
LIN {X 0.029,Y -183.492,Z 1724.106,A 0.000,B 0.000,C 90.000,E1 19.033} C_DIS
LIN {X 0.075,Y -179.359,Z 1724.087,A 0.000,B 0.000,C 90.000,E1 15.662} C_DIS
LIN {X 0.078,Y -175.150,Z 1724.064,A 0.000,B 0.000,C 90.000,E1 11.422} C_DIS
LIN {X -0.036,Y -171.965,Z 1724.040,A 0.000,B 0.000,C 90.000,E1 7.182} C_DIS
LIN {X -0.028,Y -169.443,Z 1724.011,A 0.000,B 0.000,C 90.000,E1 2.007} C_DIS
LIN {X 0.027,Y -168.431,Z 1723.969,A 0.000,B 0.000,C 90.000,E1 354.318} C_DIS
LIN {X 0.036,Y -170.277,Z 1723.920,A 0.000,B 0.000,C 90.000,E1 345.644} C_DIS
LIN {X -0.051,Y -173.060,Z 1723.892,A 0.000,B 0.000,C 90.000,E1 340.496} C_DIS
LIN {X 0.052,Y -176.531,Z 1723.868,A 0.000,B 0.000,C 90.000,E1 336.177} C_DIS
LIN {X -0.011,Y -180.890,Z 1723.844,A 0.000,B 0.000,C 90.000,E1 331.948} C_DIS
LIN {X -0.024,Y -185.256,Z 1723.825,A 0.000,B 0.000,C 90.000,E1 328.584} C_DIS
LIN {X -0.061,Y -190.576,Z 1723.807,A 0.000,B 0.000,C 90.000,E1 325.261} C_DIS
LIN {X 0.021,Y -195.300,Z 1723.793,A 0.000,B 0.000,C 90.000,E1 322.763} C_DIS
LIN {X 0.030,Y -201.712,Z 1723.777,A 0.000,B 0.000,C 90.000,E1 319.908} C_DIS
LIN {X 0.012,Y -209.055,Z 1723.762,A 0.000,B 0.000,C 90.000,E1 317.106} C_DIS
LIN {X -0.009,Y -217.461,Z 1723.746,A 0.000,B 0.000,C 90.000,E1 314.352} C_DIS
LIN {X 0.091,Y -225.562,Z 1723.734,A 0.000,B 0.000,C 90.000,E1 312.000} C_DIS
LIN {X 0.093,Y -233.135,Z 1723.723,A 0.000,B 0.000,C 90.000,E1 310.092} C_DIS
LIN {X -0.084,Y -241.573,Z 1723.712,A 0.000,B 0.000,C 90.000,E1 308.257} C_DIS
LIN {X 0.059,Y -251.082,Z 1723.702,A 0.000,B 0.000,C 90.000,E1 306.377} C_DIS
LIN {X 0.108,Y -263.840,Z 1723.690,A 0.000,B 0.000,C 90.000,E1 304.199} C_DIS
LIN {X -0.007,Y -282.378,Z 1723.675,A 0.000,B 0.000,C 90.000,E1 301.416} C_DIS
LIN {X 0.066,Y -302.259,Z 1723.659,A 0.000,B 0.000,C 90.000,E1 298.693} C_DIS
LIN {X -0.041,Y -317.754,Z 1723.649,A 0.000,B 0.000,C 90.000,E1 296.744} C_DIS
LIN {X 0.047,Y -333.454,Z 1723.638,A 0.000,B 0.000,C 90.000,E1 294.823} C_DIS
LIN {X 0.143,Y -346.447,Z 1723.629,A 0.000,B 0.000,C 90.000,E1 293.259} C_DIS
LIN {X -0.103,Y -356.637,Z 1723.623,A 0.000,B 0.000,C 90.000,E1 292.078} C_DIS
LIN {X 0.044,Y -368.944,Z 1723.614,A 0.000,B 0.000,C 90.000,E1 290.556} C_DIS
LIN {X -0.038,Y -375.946,Z 1723.609,A 0.000,B 0.000,C 90.000,E1 289.685} C_DIS
LIN {X 0.050,Y -380.217,Z 1723.606,A 0.000,B 0.000,C 90.000,E1 289.087} C_DIS
LIN {X -0.193,Y -384.062,Z 1723.603,A 0.000,B 0.000,C 90.000,E1 288.544} C_DIS
LIN {X -0.048,Y -387.524,Z 1723.600,A 0.000,B 0.000,C 90.000,E1 287.946} C_DIS
LIN {X -0.099,Y -391.871,Z 1723.595,A 0.000,B 0.000,C 90.000,E1 287.094} C_DIS
LIN {X 0.102,Y -394.220,Z 1723.592,A 0.000,B 0.000,C 90.000,E1 286.496} C_DIS
LIN {X -0.061,Y -396.235,Z 1723.589,A 0.000,B 0.000,C 90.000,E1 285.953} C_DIS
LIN {X 0.057,Y -397.867,Z 1723.585,A 0.000,B 0.000,C 90.000,E1 285.371} C_DIS
LIN {X -0.090,Y -399.130,Z 1723.582,A 0.000,B 0.000,C 90.000,E1 284.828} C_DIS
LIN {X 0.056,Y -400.011,Z 1723.579,A 0.000,B 0.000,C 90.000,E1 284.245} C_DIS
LIN {X -0.080,Y -400.549,Z 1723.576,A 0.000,B 0.000,C 90.000,E1 283.703} C_DIS
LIN {X 0.083,Y -400.682,Z 1723.573,A 0.000,B 0.000,C 90.000,E1 283.119} C_DIS
LIN {X -0.140,Y -400.405,Z 1723.570,A 0.000,B 0.000,C 90.000,E1 282.591} C_DIS
LIN {X 0.030,Y -399.699,Z 1723.567,A 0.000,B 0.000,C 90.000,E1 282.007} C_DIS
LIN {X -0.193,Y -398.560,Z 1723.564,A 0.000,B 0.000,C 90.000,E1 281.478} C_DIS
LIN {X -0.030,Y -396.875,Z 1723.561,A 0.000,B 0.000,C 90.000,E1 280.894} C_DIS
LIN {X 0.125,Y -394.633,Z 1723.557,A 0.000,B 0.000,C 90.000,E1 280.310} C_DIS
LIN {X -0.127,Y -391.790,Z 1723.554,A 0.000,B 0.000,C 90.000,E1 279.782} C_DIS
LIN {X 0.075,Y -380.067,Z 1723.543,A 0.000,B 0.000,C 90.000,E1 277.757} C_DIS
LIN {X 0.081,Y -374.546,Z 1723.538,A 0.000,B 0.000,C 90.000,E1 276.891} C_DIS
LIN {X 0.043,Y -370.209,Z 1723.535,A 0.000,B 0.000,C 90.000,E1 276.315} C_DIS
LIN {X -0.017,Y -365.186,Z 1723.532,A 0.000,B 0.000,C 90.000,E1 275.739} C_DIS
LIN {X -0.097,Y -359.497,Z 1723.529,A 0.000,B 0.000,C 90.000,E1 275.163} C_DIS
LIN {X 0.083,Y -353.523,Z 1723.526,A 0.000,B 0.000,C 90.000,E1 274.588} C_DIS
LIN {X 0.137,Y -347.335,Z 1723.523,A 0.000,B 0.000,C 90.000,E1 274.073} C_DIS
LIN {X 0.168,Y -341.099,Z 1723.520,A 0.000,B 0.000,C 90.000,E1 273.612} C_DIS
LIN {X 0.058,Y -334.711,Z 1723.518,A 0.000,B 0.000,C 90.000,E1 273.212} C_DIS
LIN {X 0.164,Y -328.070,Z 1723.516,A 0.000,B 0.000,C 90.000,E1 272.808} C_DIS
LIN {X 0.151,Y -321.461,Z 1723.514,A 0.000,B 0.000,C 90.000,E1 272.465} C_DIS
LIN {X -0.014,Y -314.385,Z 1723.512,A 0.000,B 0.000,C 90.000,E1 272.178} C_DIS
LIN {X 0.107,Y -307.380,Z 1723.511,A 0.000,B 0.000,C 90.000,E1 271.892} C_DIS
LIN {X -0.086,Y -296.821,Z 1723.509,A 0.000,B 0.000,C 90.000,E1 271.604} C_DIS
LIN {X -0.140,Y -289.497,Z 1723.508,A 0.000,B 0.000,C 90.000,E1 271.432} C_DIS
LIN {X -0.125,Y -276.987,Z 1723.507,A 0.000,B 0.000,C 90.000,E1 271.203} C_DIS
LIN {X -0.121,Y -260.039,Z 1723.505,A 0.000,B 0.000,C 90.000,E1 270.974} C_DIS
LIN {X -0.015,Y -247.433,Z 1723.505,A 0.000,B 0.000,C 90.000,E1 270.859} C_DIS
LIN {X -0.070,Y -240.336,Z 1723.505,A 0.000,B 0.000,C 90.000,E1 270.859} C_DIS
LIN {X -0.079,Y -181.494,Z 1723.505,A 0.000,B 0.000,C 90.000,E1 270.859} C_DIS
LIN {X -0.081,Y -181.519,Z 1723.499,A 0.000,B 0.000,C 90.000,E1 269.828} C_DIS
LIN {X 0.043,Y -180.906,Z 1723.475,A 0.000,B 0.000,C 90.000,E1 265.412} C_DIS
LIN {X -0.081,Y -180.716,Z 1723.470,A 0.000,B 0.000,C 90.000,E1 264.609} C_DIS
LIN {X 0.017,Y -178.804,Z 1723.442,A 0.000,B 0.000,C 90.000,E1 259.511} C_DIS
LIN {X 0.093,Y -175.849,Z 1723.413,A 0.000,B 0.000,C 90.000,E1 254.393} C_DIS
LIN {X 0.053,Y -172.584,Z 1723.390,A 0.000,B 0.000,C 90.000,E1 250.134} C_DIS
LIN {X 0.069,Y -171.474,Z 1723.380,A 0.000,B 0.000,C 90.000,E1 248.411} C_DIS
LIN {X 0.048,Y -167.704,Z 1723.356,A 0.000,B 0.000,C 90.000,E1 244.101} C_DIS
LIN {X 0.061,Y -166.392,Z 1723.347,A 0.000,B 0.000,C 90.000,E1 242.359} C_DIS
LIN {X 0.053,Y -163.117,Z 1723.327,A 0.000,B 0.000,C 90.000,E1 238.869} C_DIS
LIN {X 0.103,Y -161.067,Z 1723.313,A 0.000,B 0.000,C 90.000,E1 236.215} C_DIS
LIN {X -0.010,Y -157.801,Z 1723.293,A 0.000,B 0.000,C 90.000,E1 232.718} C_DIS
LIN {X -0.072,Y -155.836,Z 1723.278,A 0.000,B 0.000,C 90.000,E1 230.070} C_DIS
LIN {X -0.014,Y -152.087,Z 1723.253,A 0.000,B 0.000,C 90.000,E1 225.567} C_DIS
LIN {X 0.004,Y -150.337,Z 1723.238,A 0.000,B 0.000,C 90.000,E1 222.852} C_DIS
LIN {X 0.025,Y -147.076,Z 1723.213,A 0.000,B 0.000,C 90.000,E1 218.302} C_DIS
LIN {X -0.071,Y -145.650,Z 1723.198,A 0.000,B 0.000,C 90.000,E1 215.598} C_DIS
LIN {X -0.067,Y -143.032,Z 1723.172,A 0.000,B 0.000,C 90.000,E1 211.003} C_DIS
LIN {X 0.059,Y -141.657,Z 1723.152,A 0.000,B 0.000,C 90.000,E1 207.257} C_DIS
LIN {X -0.021,Y -139.447,Z 1723.115,A 0.000,B 0.000,C 90.000,E1 200.791} C_DIS
LIN {X 0.031,Y -139.180,Z 1723.105,A 0.000,B 0.000,C 90.000,E1 198.906} C_DIS
LIN {X 0.060,Y -138.320,Z 1723.053,A 0.000,B 0.000,C 90.000,E1 189.557} C_DIS
LIN {X 0.069,Y -139.465,Z 1723.006,A 0.000,B 0.000,C 90.000,E1 181.146} C_DIS
LIN {X 0.010,Y -141.029,Z 1722.975,A 0.000,B 0.000,C 90.000,E1 175.584} C_DIS
LIN {X -0.036,Y -142.396,Z 1722.960,A 0.000,B 0.000,C 90.000,E1 172.818} C_DIS
LIN {X 0.026,Y -144.628,Z 1722.934,A 0.000,B 0.000,C 90.000,E1 168.173} C_DIS
LIN {X -0.055,Y -147.823,Z 1722.909,A 0.000,B 0.000,C 90.000,E1 163.614} C_DIS
LIN {X 0.032,Y -150.514,Z 1722.889,A 0.000,B 0.000,C 90.000,E1 159.934} C_DIS
LIN {X 0.052,Y -153.976,Z 1722.869,A 0.000,B 0.000,C 90.000,E1 156.305} C_DIS
LIN {X -0.027,Y -157.387,Z 1722.849,A 0.000,B 0.000,C 90.000,E1 152.743} C_DIS
LIN {X -0.085,Y -161.592,Z 1722.829,A 0.000,B 0.000,C 90.000,E1 149.203} C_DIS
LIN {X -0.074,Y -165.788,Z 1722.809,A 0.000,B 0.000,C 90.000,E1 145.674} C_DIS
LIN {X -0.089,Y -170.750,Z 1722.790,A 0.000,B 0.000,C 90.000,E1 142.190} C_DIS
LIN {X 0.069,Y -175.622,Z 1722.771,A 0.000,B 0.000,C 90.000,E1 138.690} C_DIS
LIN {X -0.062,Y -181.238,Z 1722.752,A 0.000,B 0.000,C 90.000,E1 135.324} C_DIS
LIN {X 0.069,Y -186.708,Z 1722.733,A 0.000,B 0.000,C 90.000,E1 131.919} C_DIS
LIN {X 0.021,Y -191.307,Z 1722.719,A 0.000,B 0.000,C 90.000,E1 129.439} C_DIS
LIN {X -0.048,Y -197.136,Z 1722.701,A 0.000,B 0.000,C 90.000,E1 126.171} C_DIS
LIN {X -0.012,Y -200.412,Z 1722.692,A 0.000,B 0.000,C 90.000,E1 124.532} C_DIS
LIN {X -0.112,Y -206.296,Z 1722.674,A 0.000,B 0.000,C 90.000,E1 121.337} C_DIS
LIN {X 0.007,Y -209.659,Z 1722.665,A 0.000,B 0.000,C 90.000,E1 119.667} C_DIS
LIN {X -0.039,Y -333.451,Z 1722.665,A 0.000,B 0.000,C 90.000,E1 119.667} C_DIS
LIN {X -0.090,Y -334.519,Z 1722.665,A 0.000,B 0.000,C 90.000,E1 119.667} C_DIS
LIN {X 0.041,Y -339.718,Z 1722.664,A 0.000,B 0.000,C 90.000,E1 119.461} C_DIS
LIN {X 0.008,Y -342.266,Z 1722.663,A 0.000,B 0.000,C 90.000,E1 119.283} C_DIS
LIN {X -0.193,Y -345.666,Z 1722.661,A 0.000,B 0.000,C 90.000,E1 118.949} C_DIS
LIN {X 0.073,Y -347.572,Z 1722.659,A 0.000,B 0.000,C 90.000,E1 118.615} C_DIS
LIN {X 0.043,Y -350.423,Z 1722.656,A 0.000,B 0.000,C 90.000,E1 118.025} C_DIS
LIN {X -0.107,Y -363.498,Z 1722.641,A 0.000,B 0.000,C 90.000,E1 115.335} C_DIS
LIN {X 0.147,Y -378.106,Z 1722.626,A 0.000,B 0.000,C 90.000,E1 112.642} C_DIS
LIN {X 0.014,Y -392.483,Z 1722.613,A 0.000,B 0.000,C 90.000,E1 110.355} C_DIS
LIN {X -0.048,Y -408.272,Z 1722.601,A 0.000,B 0.000,C 90.000,E1 108.109} C_DIS
LIN {X 0.030,Y -425.582,Z 1722.588,A 0.000,B 0.000,C 90.000,E1 105.898} C_DIS
LIN {X -0.090,Y -444.515,Z 1722.576,A 0.000,B 0.000,C 90.000,E1 103.772} C_DIS
LIN {X -0.193,Y -464.495,Z 1722.565,A 0.000,B 0.000,C 90.000,E1 101.771} C_DIS
LIN {X 0.032,Y -487.634,Z 1722.554,A 0.000,B 0.000,C 90.000,E1 99.670} C_DIS
LIN {X 0.249,Y -506.025,Z 1722.546,A 0.000,B 0.000,C 90.000,E1 98.163} C_DIS
LIN {X -0.054,Y -508.421,Z 1722.544,A 0.000,B 0.000,C 90.000,E1 97.992} C_DIS
LIN {X 0.181,Y -511.806,Z 1722.542,A 0.000,B 0.000,C 90.000,E1 97.530} C_DIS
LIN {X 0.130,Y -513.031,Z 1722.541,A 0.000,B 0.000,C 90.000,E1 97.296} C_DIS
LIN {X 0.014,Y -513.918,Z 1722.539,A 0.000,B 0.000,C 90.000,E1 97.068} C_DIS
LIN {X -0.129,Y -514.830,Z 1722.537,A 0.000,B 0.000,C 90.000,E1 96.606} C_DIS
LIN {X -0.266,Y -514.715,Z 1722.534,A 0.000,B 0.000,C 90.000,E1 96.144} C_DIS
LIN {X 0.111,Y -513.550,Z 1722.531,A 0.000,B 0.000,C 90.000,E1 95.625} C_DIS
LIN {X 0.068,Y -512.517,Z 1722.530,A 0.000,B 0.000,C 90.000,E1 95.391} C_DIS
LIN {X -0.023,Y -511.111,Z 1722.529,A 0.000,B 0.000,C 90.000,E1 95.163} C_DIS
LIN {X -0.179,Y -498.462,Z 1722.519,A 0.000,B 0.000,C 90.000,E1 93.498} C_DIS
LIN {X 0.047,Y -487.633,Z 1722.511,A 0.000,B 0.000,C 90.000,E1 92.007} C_DIS
LIN {X -0.088,Y -474.855,Z 1722.502,A 0.000,B 0.000,C 90.000,E1 90.286} C_DIS
LIN {X 0.190,Y -463.890,Z 1722.493,A 0.000,B 0.000,C 90.000,E1 88.740} C_DIS
LIN {X -0.166,Y -449.186,Z 1722.482,A 0.000,B 0.000,C 90.000,E1 86.731} C_DIS
LIN {X 0.038,Y -434.457,Z 1722.470,A 0.000,B 0.000,C 90.000,E1 84.609} C_DIS
LIN {X 0.017,Y -419.771,Z 1722.458,A 0.000,B 0.000,C 90.000,E1 82.470} C_DIS
LIN {X -0.023,Y -400.467,Z 1722.441,A 0.000,B 0.000,C 90.000,E1 79.454} C_DIS
LIN {X -0.108,Y -384.013,Z 1722.426,A 0.000,B 0.000,C 90.000,E1 76.645} C_DIS
LIN {X -0.026,Y -369.781,Z 1722.411,A 0.000,B 0.000,C 90.000,E1 74.031} C_DIS
LIN {X 0.167,Y -357.432,Z 1722.398,A 0.000,B 0.000,C 90.000,E1 71.638} C_DIS
LIN {X -0.009,Y -342.680,Z 1722.381,A 0.000,B 0.000,C 90.000,E1 68.646} C_DIS
LIN {X 0.001,Y -332.636,Z 1722.369,A 0.000,B 0.000,C 90.000,E1 66.485} C_DIS
LIN {X 0.030,Y -318.610,Z 1722.352,A 0.000,B 0.000,C 90.000,E1 63.332} C_DIS
LIN {X -0.063,Y -309.018,Z 1722.339,A 0.000,B 0.000,C 90.000,E1 61.101} C_DIS
LIN {X 0.082,Y -298.094,Z 1722.325,A 0.000,B 0.000,C 90.000,E1 58.456} C_DIS
LIN {X -0.128,Y -289.879,Z 1722.314,A 0.000,B 0.000,C 90.000,E1 56.501} C_DIS
LIN {X -0.046,Y -280.125,Z 1722.301,A 0.000,B 0.000,C 90.000,E1 54.116} C_DIS
LIN {X 0.060,Y -271.698,Z 1722.289,A 0.000,B 0.000,C 90.000,E1 52.029} C_DIS
LIN {X 0.031,Y -261.961,Z 1722.276,A 0.000,B 0.000,C 90.000,E1 49.585} C_DIS
LIN {X 0.122,Y -252.384,Z 1722.262,A 0.000,B 0.000,C 90.000,E1 47.067} C_DIS
LIN {X 0.131,Y -240.538,Z 1722.243,A 0.000,B 0.000,C 90.000,E1 43.785} C_DIS
LIN {X -0.001,Y -229.442,Z 1722.225,A 0.000,B 0.000,C 90.000,E1 40.458} C_DIS
LIN {X -0.057,Y -221.573,Z 1722.210,A 0.000,B 0.000,C 90.000,E1 37.810} C_DIS
LIN {X 0.049,Y -213.303,Z 1722.193,A 0.000,B 0.000,C 90.000,E1 34.692} C_DIS
LIN {X 0.059,Y -205.889,Z 1722.175,A 0.000,B 0.000,C 90.000,E1 31.544} C_DIS
LIN {X 0.023,Y -199.126,Z 1722.158,A 0.000,B 0.000,C 90.000,E1 28.359} C_DIS
LIN {X -0.107,Y -193.051,Z 1722.140,A 0.000,B 0.000,C 90.000,E1 25.155} C_DIS
LIN {X -0.019,Y -187.488,Z 1722.121,A 0.000,B 0.000,C 90.000,E1 21.844} C_DIS
LIN {X -0.100,Y -182.695,Z 1722.103,A 0.000,B 0.000,C 90.000,E1 18.544} C_DIS
LIN {X 0.049,Y -178.706,Z 1722.084,A 0.000,B 0.000,C 90.000,E1 15.134} C_DIS
LIN {X 0.035,Y -174.617,Z 1722.061,A 0.000,B 0.000,C 90.000,E1 10.894} C_DIS
LIN {X 0.049,Y -171.524,Z 1722.037,A 0.000,B 0.000,C 90.000,E1 6.606} C_DIS
LIN {X 0.038,Y -169.174,Z 1722.008,A 0.000,B 0.000,C 90.000,E1 1.432} C_DIS
LIN {X 0.023,Y -168.318,Z 1721.969,A 0.000,B 0.000,C 90.000,E1 354.318} C_DIS
LIN {X -0.004,Y -169.842,Z 1721.925,A 0.000,B 0.000,C 90.000,E1 346.520} C_DIS
LIN {X 0.020,Y -172.434,Z 1721.896,A 0.000,B 0.000,C 90.000,E1 341.329} C_DIS
LIN {X -0.018,Y -175.712,Z 1721.872,A 0.000,B 0.000,C 90.000,E1 337.050} C_DIS
LIN {X -0.026,Y -179.908,Z 1721.849,A 0.000,B 0.000,C 90.000,E1 332.794} C_DIS
LIN {X 0.002,Y -184.088,Z 1721.830,A 0.000,B 0.000,C 90.000,E1 329.410} C_DIS
LIN {X -0.066,Y -189.178,Z 1721.812,A 0.000,B 0.000,C 90.000,E1 326.087} C_DIS
LIN {X 0.031,Y -193.691,Z 1721.798,A 0.000,B 0.000,C 90.000,E1 323.577} C_DIS
LIN {X 0.014,Y -198.919,Z 1721.784,A 0.000,B 0.000,C 90.000,E1 321.126} C_DIS
LIN {X -0.075,Y -205.909,Z 1721.768,A 0.000,B 0.000,C 90.000,E1 318.324} C_DIS
LIN {X 0.095,Y -212.674,Z 1721.755,A 0.000,B 0.000,C 90.000,E1 315.891} C_DIS
LIN {X 0.008,Y -221.564,Z 1721.740,A 0.000,B 0.000,C 90.000,E1 313.176} C_DIS
LIN {X 0.040,Y -230.207,Z 1721.727,A 0.000,B 0.000,C 90.000,E1 310.862} C_DIS
LIN {X -0.033,Y -238.275,Z 1721.717,A 0.000,B 0.000,C 90.000,E1 308.991} C_DIS
LIN {X -0.139,Y -247.358,Z 1721.706,A 0.000,B 0.000,C 90.000,E1 307.156} C_DIS
LIN {X -0.141,Y -261.805,Z 1721.692,A 0.000,B 0.000,C 90.000,E1 304.612} C_DIS
LIN {X -0.117,Y -277.867,Z 1721.678,A 0.000,B 0.000,C 90.000,E1 302.133} C_DIS
LIN {X 0.080,Y -299.892,Z 1721.661,A 0.000,B 0.000,C 90.000,E1 299.027} C_DIS
LIN {X -0.022,Y -317.909,Z 1721.649,A 0.000,B 0.000,C 90.000,E1 296.744} C_DIS
LIN {X 0.045,Y -333.608,Z 1721.638,A 0.000,B 0.000,C 90.000,E1 294.823} C_DIS
LIN {X 0.100,Y -346.616,Z 1721.629,A 0.000,B 0.000,C 90.000,E1 293.259} C_DIS
LIN {X 0.004,Y -359.151,Z 1721.621,A 0.000,B 0.000,C 90.000,E1 291.770} C_DIS
LIN {X -0.144,Y -371.359,Z 1721.613,A 0.000,B 0.000,C 90.000,E1 290.301} C_DIS
LIN {X 0.012,Y -378.170,Z 1721.608,A 0.000,B 0.000,C 90.000,E1 289.396} C_DIS
LIN {X -0.120,Y -382.261,Z 1721.604,A 0.000,B 0.000,C 90.000,E1 288.833} C_DIS
LIN {X 0.031,Y -387.615,Z 1721.600,A 0.000,B 0.000,C 90.000,E1 287.946} C_DIS
LIN {X -0.018,Y -392.012,Z 1721.595,A 0.000,B 0.000,C 90.000,E1 287.094} C_DIS
LIN {X 0.184,Y -394.394,Z 1721.592,A 0.000,B 0.000,C 90.000,E1 286.496} C_DIS
LIN {X -0.087,Y -396.418,Z 1721.589,A 0.000,B 0.000,C 90.000,E1 285.969} C_DIS
LIN {X 0.142,Y -398.041,Z 1721.585,A 0.000,B 0.000,C 90.000,E1 285.371} C_DIS
LIN {X -0.004,Y -399.327,Z 1721.582,A 0.000,B 0.000,C 90.000,E1 284.828} C_DIS
LIN {X 0.144,Y -400.236,Z 1721.579,A 0.000,B 0.000,C 90.000,E1 284.245} C_DIS
LIN {X 0.008,Y -400.794,Z 1721.576,A 0.000,B 0.000,C 90.000,E1 283.703} C_DIS
LIN {X 0.173,Y -400.940,Z 1721.573,A 0.000,B 0.000,C 90.000,E1 283.119} C_DIS
LIN {X -0.049,Y -400.666,Z 1721.570,A 0.000,B 0.000,C 90.000,E1 282.591} C_DIS
LIN {X 0.122,Y -399.944,Z 1721.567,A 0.000,B 0.000,C 90.000,E1 282.007} C_DIS
LIN {X -0.099,Y -398.769,Z 1721.564,A 0.000,B 0.000,C 90.000,E1 281.478} C_DIS
LIN {X 0.065,Y -397.093,Z 1721.561,A 0.000,B 0.000,C 90.000,E1 280.894} C_DIS
LIN {X -0.168,Y -394.858,Z 1721.557,A 0.000,B 0.000,C 90.000,E1 280.366} C_DIS
LIN {X -0.097,Y -392.042,Z 1721.554,A 0.000,B 0.000,C 90.000,E1 279.792} C_DIS
LIN {X 0.147,Y -381.946,Z 1721.545,A 0.000,B 0.000,C 90.000,E1 278.049} C_DIS
LIN {X 0.166,Y -376.669,Z 1721.540,A 0.000,B 0.000,C 90.000,E1 277.182} C_DIS
LIN {X 0.139,Y -372.618,Z 1721.537,A 0.000,B 0.000,C 90.000,E1 276.606} C_DIS
LIN {X 0.092,Y -367.960,Z 1721.534,A 0.000,B 0.000,C 90.000,E1 276.030} C_DIS
LIN {X 0.027,Y -362.622,Z 1721.530,A 0.000,B 0.000,C 90.000,E1 275.454} C_DIS
LIN {X 0.082,Y -356.819,Z 1721.527,A 0.000,B 0.000,C 90.000,E1 274.878} C_DIS
LIN {X 0.050,Y -350.810,Z 1721.524,A 0.000,B 0.000,C 90.000,E1 274.359} C_DIS
LIN {X -0.047,Y -344.577,Z 1721.522,A 0.000,B 0.000,C 90.000,E1 273.898} C_DIS
LIN {X -0.097,Y -335.081,Z 1721.518,A 0.000,B 0.000,C 90.000,E1 273.269} C_DIS
LIN {X 0.013,Y -325.166,Z 1721.515,A 0.000,B 0.000,C 90.000,E1 272.694} C_DIS
LIN {X 0.108,Y -318.465,Z 1721.513,A 0.000,B 0.000,C 90.000,E1 272.350} C_DIS
LIN {X 0.093,Y -311.436,Z 1721.512,A 0.000,B 0.000,C 90.000,E1 272.064} C_DIS
LIN {X 0.009,Y -300.672,Z 1721.510,A 0.000,B 0.000,C 90.000,E1 271.718} C_DIS
LIN {X -0.123,Y -293.575,Z 1721.508,A 0.000,B 0.000,C 90.000,E1 271.547} C_DIS
LIN {X 0.077,Y -281.924,Z 1721.507,A 0.000,B 0.000,C 90.000,E1 271.260} C_DIS
LIN {X -0.030,Y -264.870,Z 1721.506,A 0.000,B 0.000,C 90.000,E1 271.031} C_DIS
LIN {X -0.110,Y -251.202,Z 1721.505,A 0.000,B 0.000,C 90.000,E1 270.917} C_DIS
LIN {X 0.055,Y -244.759,Z 1721.505,A 0.000,B 0.000,C 90.000,E1 270.859} C_DIS
LIN {X 0.026,Y -234.217,Z 1721.505,A 0.000,B 0.000,C 90.000,E1 270.859} C_DIS
LIN {X -0.006,Y -181.488,Z 1721.505,A 0.000,B 0.000,C 90.000,E1 270.859} C_DIS
LIN {X -0.009,Y -181.525,Z 1721.499,A 0.000,B 0.000,C 90.000,E1 269.828} C_DIS
LIN {X -0.066,Y -180.907,Z 1721.475,A 0.000,B 0.000,C 90.000,E1 265.469} C_DIS
LIN {X -0.009,Y -180.727,Z 1721.470,A 0.000,B 0.000,C 90.000,E1 264.609} C_DIS
LIN {X 0.089,Y -178.816,Z 1721.442,A 0.000,B 0.000,C 90.000,E1 259.511} C_DIS
LIN {X -0.005,Y -175.861,Z 1721.414,A 0.000,B 0.000,C 90.000,E1 254.448} C_DIS
LIN {X 0.043,Y -173.827,Z 1721.399,A 0.000,B 0.000,C 90.000,E1 251.873} C_DIS
LIN {X -0.021,Y -171.494,Z 1721.380,A 0.000,B 0.000,C 90.000,E1 248.465} C_DIS
LIN {X -0.034,Y -167.722,Z 1721.356,A 0.000,B 0.000,C 90.000,E1 244.152} C_DIS
LIN {X -0.018,Y -166.415,Z 1721.347,A 0.000,B 0.000,C 90.000,E1 242.410} C_DIS
LIN {X -0.019,Y -163.137,Z 1721.327,A 0.000,B 0.000,C 90.000,E1 238.918} C_DIS
LIN {X -0.054,Y -161.091,Z 1721.313,A 0.000,B 0.000,C 90.000,E1 236.294} C_DIS
LIN {X -0.070,Y -157.820,Z 1721.293,A 0.000,B 0.000,C 90.000,E1 232.763} C_DIS
LIN {X -0.006,Y -155.854,Z 1721.278,A 0.000,B 0.000,C 90.000,E1 230.070} C_DIS
LIN {X 0.050,Y -152.104,Z 1721.253,A 0.000,B 0.000,C 90.000,E1 225.567} C_DIS
LIN {X 0.068,Y -150.355,Z 1721.238,A 0.000,B 0.000,C 90.000,E1 222.852} C_DIS
LIN {X -0.003,Y -147.091,Z 1721.213,A 0.000,B 0.000,C 90.000,E1 218.338} C_DIS
LIN {X -0.008,Y -145.662,Z 1721.198,A 0.000,B 0.000,C 90.000,E1 215.598} C_DIS
LIN {X -0.005,Y -143.044,Z 1721.172,A 0.000,B 0.000,C 90.000,E1 211.003} C_DIS
LIN {X -0.005,Y -141.668,Z 1721.152,A 0.000,B 0.000,C 90.000,E1 207.308} C_DIS
LIN {X 0.040,Y -139.451,Z 1721.116,A 0.000,B 0.000,C 90.000,E1 200.791} C_DIS
LIN {X -0.039,Y -139.185,Z 1721.105,A 0.000,B 0.000,C 90.000,E1 198.960} C_DIS
LIN {X -0.016,Y -138.322,Z 1721.053,A 0.000,B 0.000,C 90.000,E1 189.613} C_DIS
LIN {X -0.009,Y -139.462,Z 1721.007,A 0.000,B 0.000,C 90.000,E1 181.203} C_DIS
LIN {X -0.069,Y -141.018,Z 1720.976,A 0.000,B 0.000,C 90.000,E1 175.641} C_DIS
LIN {X 0.027,Y -142.382,Z 1720.960,A 0.000,B 0.000,C 90.000,E1 172.818} C_DIS
LIN {X -0.052,Y -144.613,Z 1720.934,A 0.000,B 0.000,C 90.000,E1 168.229} C_DIS
LIN {X 0.010,Y -147.807,Z 1720.909,A 0.000,B 0.000,C 90.000,E1 163.614} C_DIS
LIN {X 0.045,Y -150.494,Z 1720.889,A 0.000,B 0.000,C 90.000,E1 159.953} C_DIS
LIN {X -0.024,Y -153.950,Z 1720.869,A 0.000,B 0.000,C 90.000,E1 156.357} C_DIS
LIN {X 0.040,Y -157.362,Z 1720.849,A 0.000,B 0.000,C 90.000,E1 152.743} C_DIS
LIN {X -0.018,Y -161.560,Z 1720.829,A 0.000,B 0.000,C 90.000,E1 149.203} C_DIS
LIN {X -0.005,Y -165.757,Z 1720.809,A 0.000,B 0.000,C 90.000,E1 145.674} C_DIS
LIN {X -0.019,Y -170.713,Z 1720.790,A 0.000,B 0.000,C 90.000,E1 142.190} C_DIS
LIN {X 0.024,Y -175.586,Z 1720.771,A 0.000,B 0.000,C 90.000,E1 138.728} C_DIS
LIN {X 0.011,Y -181.204,Z 1720.752,A 0.000,B 0.000,C 90.000,E1 135.324} C_DIS
LIN {X 0.004,Y -186.667,Z 1720.733,A 0.000,B 0.000,C 90.000,E1 131.962} C_DIS
LIN {X -0.052,Y -191.271,Z 1720.719,A 0.000,B 0.000,C 90.000,E1 129.483} C_DIS
LIN {X 0.028,Y -197.094,Z 1720.701,A 0.000,B 0.000,C 90.000,E1 126.171} C_DIS
LIN {X 0.064,Y -200.368,Z 1720.692,A 0.000,B 0.000,C 90.000,E1 124.532} C_DIS
LIN {X -0.034,Y -206.254,Z 1720.674,A 0.000,B 0.000,C 90.000,E1 121.337} C_DIS
LIN {X 0.086,Y -209.613,Z 1720.665,A 0.000,B 0.000,C 90.000,E1 119.667} C_DIS
LIN {X 0.086,Y -334.247,Z 1720.665,A 0.000,B 0.000,C 90.000,E1 119.667} C_DIS
LIN {X 0.002,Y -339.688,Z 1720.664,A 0.000,B 0.000,C 90.000,E1 119.489} C_DIS
LIN {X 0.136,Y -342.201,Z 1720.663,A 0.000,B 0.000,C 90.000,E1 119.283} C_DIS
LIN {X -0.064,Y -345.572,Z 1720.661,A 0.000,B 0.000,C 90.000,E1 118.949} C_DIS
LIN {X 0.192,Y -347.475,Z 1720.659,A 0.000,B 0.000,C 90.000,E1 118.615} C_DIS
LIN {X 0.152,Y -350.320,Z 1720.656,A 0.000,B 0.000,C 90.000,E1 118.025} C_DIS
LIN {X 0.003,Y -363.386,Z 1720.641,A 0.000,B 0.000,C 90.000,E1 115.335} C_DIS
LIN {X -0.091,Y -377.983,Z 1720.626,A 0.000,B 0.000,C 90.000,E1 112.695} C_DIS
LIN {X -0.010,Y -392.350,Z 1720.613,A 0.000,B 0.000,C 90.000,E1 110.375} C_DIS
LIN {X -0.062,Y -408.129,Z 1720.601,A 0.000,B 0.000,C 90.000,E1 108.127} C_DIS
LIN {X 0.144,Y -425.427,Z 1720.588,A 0.000,B 0.000,C 90.000,E1 105.898} C_DIS
LIN {X 0.025,Y -444.349,Z 1720.577,A 0.000,B 0.000,C 90.000,E1 103.772} C_DIS
LIN {X -0.083,Y -464.325,Z 1720.565,A 0.000,B 0.000,C 90.000,E1 101.771} C_DIS
LIN {X 0.136,Y -487.460,Z 1720.554,A 0.000,B 0.000,C 90.000,E1 99.670} C_DIS
LIN {X -0.153,Y -505.847,Z 1720.546,A 0.000,B 0.000,C 90.000,E1 98.219} C_DIS
LIN {X 0.044,Y -508.231,Z 1720.544,A 0.000,B 0.000,C 90.000,E1 97.992} C_DIS
LIN {X 0.189,Y -510.143,Z 1720.543,A 0.000,B 0.000,C 90.000,E1 97.757} C_DIS
LIN {X -0.242,Y -511.606,Z 1720.542,A 0.000,B 0.000,C 90.000,E1 97.587} C_DIS
LIN {X 0.220,Y -512.821,Z 1720.541,A 0.000,B 0.000,C 90.000,E1 97.296} C_DIS
LIN {X 0.108,Y -513.699,Z 1720.539,A 0.000,B 0.000,C 90.000,E1 97.068} C_DIS
LIN {X -0.035,Y -514.604,Z 1720.537,A 0.000,B 0.000,C 90.000,E1 96.606} C_DIS
LIN {X -0.174,Y -514.481,Z 1720.534,A 0.000,B 0.000,C 90.000,E1 96.144} C_DIS
LIN {X 0.202,Y -513.308,Z 1720.531,A 0.000,B 0.000,C 90.000,E1 95.625} C_DIS
LIN {X 0.158,Y -512.268,Z 1720.530,A 0.000,B 0.000,C 90.000,E1 95.391} C_DIS
LIN {X 0.065,Y -510.857,Z 1720.529,A 0.000,B 0.000,C 90.000,E1 95.163} C_DIS
LIN {X -0.096,Y -498.209,Z 1720.519,A 0.000,B 0.000,C 90.000,E1 93.498} C_DIS
LIN {X 0.123,Y -487.362,Z 1720.511,A 0.000,B 0.000,C 90.000,E1 92.007} C_DIS
LIN {X -0.019,Y -474.602,Z 1720.502,A 0.000,B 0.000,C 90.000,E1 90.286} C_DIS
LIN {X -0.211,Y -463.629,Z 1720.493,A 0.000,B 0.000,C 90.000,E1 88.797} C_DIS
LIN {X -0.112,Y -448.914,Z 1720.482,A 0.000,B 0.000,C 90.000,E1 86.731} C_DIS
LIN {X 0.084,Y -434.163,Z 1720.470,A 0.000,B 0.000,C 90.000,E1 84.609} C_DIS
LIN {X 0.054,Y -419.474,Z 1720.458,A 0.000,B 0.000,C 90.000,E1 82.470} C_DIS
LIN {X 0.004,Y -400.144,Z 1720.441,A 0.000,B 0.000,C 90.000,E1 79.454} C_DIS
LIN {X -0.091,Y -383.655,Z 1720.426,A 0.000,B 0.000,C 90.000,E1 76.645} C_DIS
LIN {X -0.021,Y -369.400,Z 1720.411,A 0.000,B 0.000,C 90.000,E1 74.031} C_DIS
LIN {X 0.163,Y -357.058,Z 1720.398,A 0.000,B 0.000,C 90.000,E1 71.638} C_DIS
LIN {X -0.023,Y -342.275,Z 1720.381,A 0.000,B 0.000,C 90.000,E1 68.646} C_DIS
LIN {X -0.022,Y -332.212,Z 1720.369,A 0.000,B 0.000,C 90.000,E1 66.485} C_DIS
LIN {X -0.004,Y -318.176,Z 1720.352,A 0.000,B 0.000,C 90.000,E1 63.332} C_DIS
LIN {X 0.164,Y -308.579,Z 1720.339,A 0.000,B 0.000,C 90.000,E1 61.051} C_DIS
LIN {X 0.031,Y -297.687,Z 1720.325,A 0.000,B 0.000,C 90.000,E1 58.456} C_DIS
LIN {X -0.186,Y -289.479,Z 1720.314,A 0.000,B 0.000,C 90.000,E1 56.501} C_DIS
LIN {X -0.110,Y -279.744,Z 1720.301,A 0.000,B 0.000,C 90.000,E1 54.116} C_DIS
LIN {X -0.010,Y -271.309,Z 1720.289,A 0.000,B 0.000,C 90.000,E1 52.029} C_DIS
LIN {X -0.044,Y -261.567,Z 1720.275,A 0.000,B 0.000,C 90.000,E1 49.585} C_DIS
LIN {X 0.064,Y -250.636,Z 1720.260,A 0.000,B 0.000,C 90.000,E1 46.701} C_DIS
LIN {X 0.024,Y -238.881,Z 1720.241,A 0.000,B 0.000,C 90.000,E1 43.419} C_DIS
LIN {X -0.139,Y -227.918,Z 1720.223,A 0.000,B 0.000,C 90.000,E1 40.092} C_DIS
LIN {X 0.022,Y -219.144,Z 1720.206,A 0.000,B 0.000,C 90.000,E1 36.996} C_DIS
LIN {X -0.062,Y -211.108,Z 1720.188,A 0.000,B 0.000,C 90.000,E1 33.913} C_DIS
LIN {X 0.065,Y -203.925,Z 1720.171,A 0.000,B 0.000,C 90.000,E1 30.718} C_DIS
LIN {X 0.053,Y -197.381,Z 1720.153,A 0.000,B 0.000,C 90.000,E1 27.513} C_DIS
LIN {X 0.051,Y -191.462,Z 1720.135,A 0.000,B 0.000,C 90.000,E1 24.259} C_DIS
LIN {X 0.018,Y -186.100,Z 1720.117,A 0.000,B 0.000,C 90.000,E1 20.972} C_DIS
LIN {X 0.009,Y -181.498,Z 1720.098,A 0.000,B 0.000,C 90.000,E1 17.638} C_DIS
LIN {X 0.035,Y -176.857,Z 1720.075,A 0.000,B 0.000,C 90.000,E1 13.411} C_DIS
LIN {X 0.026,Y -173.165,Z 1720.051,A 0.000,B 0.000,C 90.000,E1 9.151} C_DIS
LIN {X -0.044,Y -170.451,Z 1720.027,A 0.000,B 0.000,C 90.000,E1 4.878} C_DIS
LIN {X -0.073,Y -168.400,Z 1719.988,A 0.000,B 0.000,C 90.000,E1 357.822} C_DIS
LIN {X -0.012,Y -169.767,Z 1719.925,A 0.000,B 0.000,C 90.000,E1 346.520} C_DIS
LIN {X 0.009,Y -172.377,Z 1719.896,A 0.000,B 0.000,C 90.000,E1 341.329} C_DIS
LIN {X -0.031,Y -175.665,Z 1719.872,A 0.000,B 0.000,C 90.000,E1 337.050} C_DIS
LIN {X -0.040,Y -179.882,Z 1719.849,A 0.000,B 0.000,C 90.000,E1 332.794} C_DIS
LIN {X -0.013,Y -184.075,Z 1719.830,A 0.000,B 0.000,C 90.000,E1 329.410} C_DIS
LIN {X -0.082,Y -189.208,Z 1719.811,A 0.000,B 0.000,C 90.000,E1 326.087} C_DIS
LIN {X 0.015,Y -193.740,Z 1719.798,A 0.000,B 0.000,C 90.000,E1 323.577} C_DIS
LIN {X -0.001,Y -199.003,Z 1719.784,A 0.000,B 0.000,C 90.000,E1 321.126} C_DIS
LIN {X -0.089,Y -206.008,Z 1719.768,A 0.000,B 0.000,C 90.000,E1 318.324} C_DIS
LIN {X 0.084,Y -212.823,Z 1719.755,A 0.000,B 0.000,C 90.000,E1 315.891} C_DIS
LIN {X -0.001,Y -221.746,Z 1719.740,A 0.000,B 0.000,C 90.000,E1 313.176} C_DIS
LIN {X 0.034,Y -230.405,Z 1719.727,A 0.000,B 0.000,C 90.000,E1 310.862} C_DIS
LIN {X -0.035,Y -238.480,Z 1719.717,A 0.000,B 0.000,C 90.000,E1 308.991} C_DIS
LIN {X -0.139,Y -247.574,Z 1719.706,A 0.000,B 0.000,C 90.000,E1 307.156} C_DIS
LIN {X -0.136,Y -262.023,Z 1719.692,A 0.000,B 0.000,C 90.000,E1 304.612} C_DIS
LIN {X 0.072,Y -280.402,Z 1719.677,A 0.000,B 0.000,C 90.000,E1 301.750} C_DIS
LIN {X -0.166,Y -300.064,Z 1719.661,A 0.000,B 0.000,C 90.000,E1 299.077} C_DIS
LIN {X -0.046,Y -315.462,Z 1719.650,A 0.000,B 0.000,C 90.000,E1 297.078} C_DIS
LIN {X -0.050,Y -331.127,Z 1719.640,A 0.000,B 0.000,C 90.000,E1 295.155} C_DIS
LIN {X -0.042,Y -344.171,Z 1719.631,A 0.000,B 0.000,C 90.000,E1 293.590} C_DIS
LIN {X 0.186,Y -356.927,Z 1719.623,A 0.000,B 0.000,C 90.000,E1 292.025} C_DIS
LIN {X 0.101,Y -369.105,Z 1719.614,A 0.000,B 0.000,C 90.000,E1 290.556} C_DIS
LIN {X 0.023,Y -376.132,Z 1719.609,A 0.000,B 0.000,C 90.000,E1 289.685} C_DIS
LIN {X 0.228,Y -382.435,Z 1719.604,A 0.000,B 0.000,C 90.000,E1 288.779} C_DIS
LIN {X 0.018,Y -387.794,Z 1719.600,A 0.000,B 0.000,C 90.000,E1 287.946} C_DIS
LIN {X -0.030,Y -392.169,Z 1719.595,A 0.000,B 0.000,C 90.000,E1 287.094} C_DIS
LIN {X 0.173,Y -394.590,Z 1719.592,A 0.000,B 0.000,C 90.000,E1 286.496} C_DIS
LIN {X -0.095,Y -396.615,Z 1719.589,A 0.000,B 0.000,C 90.000,E1 285.969} C_DIS
LIN {X 0.134,Y -398.239,Z 1719.585,A 0.000,B 0.000,C 90.000,E1 285.371} C_DIS
LIN {X -0.012,Y -399.524,Z 1719.582,A 0.000,B 0.000,C 90.000,E1 284.828} C_DIS
LIN {X 0.138,Y -400.458,Z 1719.579,A 0.000,B 0.000,C 90.000,E1 284.245} C_DIS
LIN {X 0.004,Y -401.047,Z 1719.576,A 0.000,B 0.000,C 90.000,E1 283.703} C_DIS
LIN {X 0.169,Y -401.173,Z 1719.573,A 0.000,B 0.000,C 90.000,E1 283.119} C_DIS
LIN {X -0.051,Y -400.898,Z 1719.570,A 0.000,B 0.000,C 90.000,E1 282.591} C_DIS
LIN {X 0.122,Y -400.190,Z 1719.567,A 0.000,B 0.000,C 90.000,E1 282.007} C_DIS
LIN {X -0.098,Y -399.003,Z 1719.564,A 0.000,B 0.000,C 90.000,E1 281.478} C_DIS
LIN {X 0.068,Y -397.291,Z 1719.561,A 0.000,B 0.000,C 90.000,E1 280.894} C_DIS
LIN {X -0.164,Y -395.065,Z 1719.557,A 0.000,B 0.000,C 90.000,E1 280.366} C_DIS
LIN {X -0.092,Y -392.219,Z 1719.554,A 0.000,B 0.000,C 90.000,E1 279.792} C_DIS
LIN {X 0.155,Y -382.063,Z 1719.545,A 0.000,B 0.000,C 90.000,E1 278.049} C_DIS
LIN {X 0.175,Y -376.763,Z 1719.540,A 0.000,B 0.000,C 90.000,E1 277.182} C_DIS
LIN {X 0.149,Y -372.718,Z 1719.537,A 0.000,B 0.000,C 90.000,E1 276.606} C_DIS
LIN {X 0.102,Y -368.039,Z 1719.534,A 0.000,B 0.000,C 90.000,E1 276.030} C_DIS
LIN {X 0.031,Y -362.715,Z 1719.530,A 0.000,B 0.000,C 90.000,E1 275.454} C_DIS
LIN {X 0.094,Y -356.900,Z 1719.527,A 0.000,B 0.000,C 90.000,E1 274.878} C_DIS
LIN {X 0.098,Y -350.886,Z 1719.524,A 0.000,B 0.000,C 90.000,E1 274.359} C_DIS
LIN {X 0.014,Y -344.687,Z 1719.522,A 0.000,B 0.000,C 90.000,E1 273.898} C_DIS
LIN {X -0.170,Y -338.320,Z 1719.519,A 0.000,B 0.000,C 90.000,E1 273.498} C_DIS
LIN {X -0.103,Y -331.873,Z 1719.517,A 0.000,B 0.000,C 90.000,E1 273.094} C_DIS
LIN {X 0.127,Y -325.268,Z 1719.515,A 0.000,B 0.000,C 90.000,E1 272.694} C_DIS
LIN {X -0.089,Y -318.553,Z 1719.513,A 0.000,B 0.000,C 90.000,E1 272.407} C_DIS
LIN {X -0.079,Y -311.545,Z 1719.512,A 0.000,B 0.000,C 90.000,E1 272.121} C_DIS
LIN {X -0.149,Y -304.575,Z 1719.510,A 0.000,B 0.000,C 90.000,E1 271.892} C_DIS
LIN {X 0.062,Y -294.112,Z 1719.509,A 0.000,B 0.000,C 90.000,E1 271.547} C_DIS
LIN {X -0.033,Y -282.686,Z 1719.507,A 0.000,B 0.000,C 90.000,E1 271.318} C_DIS
LIN {X 0.110,Y -269.872,Z 1719.506,A 0.000,B 0.000,C 90.000,E1 271.088} C_DIS
LIN {X -0.118,Y -256.117,Z 1719.505,A 0.000,B 0.000,C 90.000,E1 270.974} C_DIS
LIN {X -0.091,Y -244.869,Z 1719.505,A 0.000,B 0.000,C 90.000,E1 270.917} C_DIS
LIN {X -0.089,Y -181.481,Z 1719.505,A 0.000,B 0.000,C 90.000,E1 270.917} C_DIS
LIN {X 0.001,Y -181.561,Z 1719.500,A 0.000,B 0.000,C 90.000,E1 270.000} C_DIS
LIN {X -0.013,Y -180.849,Z 1719.472,A 0.000,B 0.000,C 90.000,E1 264.951} C_DIS
LIN {X 0.069,Y -178.959,Z 1719.444,A 0.000,B 0.000,C 90.000,E1 259.859} C_DIS
LIN {X -0.039,Y -177.364,Z 1719.430,A 0.000,B 0.000,C 90.000,E1 257.353} C_DIS
LIN {X 0.057,Y -175.536,Z 1719.411,A 0.000,B 0.000,C 90.000,E1 253.921} C_DIS
LIN {X 0.058,Y -172.270,Z 1719.387,A 0.000,B 0.000,C 90.000,E1 249.645} C_DIS
LIN {X 0.096,Y -171.750,Z 1719.382,A 0.000,B 0.000,C 90.000,E1 248.773} C_DIS
LIN {X -0.046,Y -167.347,Z 1719.354,A 0.000,B 0.000,C 90.000,E1 243.640} C_DIS
LIN {X 0.036,Y -166.734,Z 1719.349,A 0.000,B 0.000,C 90.000,E1 242.743} C_DIS
LIN {X -0.052,Y -162.714,Z 1719.324,A 0.000,B 0.000,C 90.000,E1 238.408} C_DIS
LIN {X 0.010,Y -161.405,Z 1719.315,A 0.000,B 0.000,C 90.000,E1 236.628} C_DIS
LIN {X 0.052,Y -157.398,Z 1719.290,A 0.000,B 0.000,C 90.000,E1 232.190} C_DIS
LIN {X -0.016,Y -155.396,Z 1719.275,A 0.000,B 0.000,C 90.000,E1 229.542} C_DIS
LIN {X -0.084,Y -151.729,Z 1719.250,A 0.000,B 0.000,C 90.000,E1 225.081} C_DIS
LIN {X -0.071,Y -149.924,Z 1719.235,A 0.000,B 0.000,C 90.000,E1 222.366} C_DIS
LIN {X -0.043,Y -146.776,Z 1719.210,A 0.000,B 0.000,C 90.000,E1 217.810} C_DIS
LIN {X 0.061,Y -145.347,Z 1719.195,A 0.000,B 0.000,C 90.000,E1 215.025} C_DIS
LIN {X -0.024,Y -142.421,Z 1719.164,A 0.000,B 0.000,C 90.000,E1 209.539} C_DIS
LIN {X 0.026,Y -141.408,Z 1719.149,A 0.000,B 0.000,C 90.000,E1 206.744} C_DIS
LIN {X 0.012,Y -139.358,Z 1719.113,A 0.000,B 0.000,C 90.000,E1 200.248} C_DIS
LIN {X 0.001,Y -138.800,Z 1719.097,A 0.000,B 0.000,C 90.000,E1 197.457} C_DIS
LIN {X 0.055,Y -138.348,Z 1719.055,A 0.000,B 0.000,C 90.000,E1 189.962} C_DIS
LIN {X -0.066,Y -139.370,Z 1719.009,A 0.000,B 0.000,C 90.000,E1 181.604} C_DIS
LIN {X -0.013,Y -141.258,Z 1718.973,A 0.000,B 0.000,C 90.000,E1 175.065} C_DIS
LIN {X -0.055,Y -142.626,Z 1718.957,A 0.000,B 0.000,C 90.000,E1 172.299} C_DIS
LIN {X 0.038,Y -144.948,Z 1718.931,A 0.000,B 0.000,C 90.000,E1 167.645} C_DIS
LIN {X 0.029,Y -147.576,Z 1718.911,A 0.000,B 0.000,C 90.000,E1 163.976} C_DIS
LIN {X -0.081,Y -150.188,Z 1718.891,A 0.000,B 0.000,C 90.000,E1 160.369} C_DIS
LIN {X -0.074,Y -153.567,Z 1718.871,A 0.000,B 0.000,C 90.000,E1 156.741} C_DIS
LIN {X -0.022,Y -156.984,Z 1718.851,A 0.000,B 0.000,C 90.000,E1 153.127} C_DIS
LIN {X 0.051,Y -161.097,Z 1718.831,A 0.000,B 0.000,C 90.000,E1 149.537} C_DIS
LIN {X -0.003,Y -163.200,Z 1718.821,A 0.000,B 0.000,C 90.000,E1 147.788} C_DIS
LIN {X 0.001,Y -167.626,Z 1718.802,A 0.000,B 0.000,C 90.000,E1 144.276} C_DIS
LIN {X 0.017,Y -171.453,Z 1718.787,A 0.000,B 0.000,C 90.000,E1 141.662} C_DIS
LIN {X -0.052,Y -176.377,Z 1718.768,A 0.000,B 0.000,C 90.000,E1 138.243} C_DIS
LIN {X 0.070,Y -180.670,Z 1718.754,A 0.000,B 0.000,C 90.000,E1 135.648} C_DIS
LIN {X 0.052,Y -186.072,Z 1718.735,A 0.000,B 0.000,C 90.000,E1 132.285} C_DIS
LIN {X -0.012,Y -190.709,Z 1718.721,A 0.000,B 0.000,C 90.000,E1 129.806} C_DIS
LIN {X 0.022,Y -196.461,Z 1718.703,A 0.000,B 0.000,C 90.000,E1 126.503} C_DIS
LIN {X -0.013,Y -201.242,Z 1718.689,A 0.000,B 0.000,C 90.000,E1 124.072} C_DIS
LIN {X -0.086,Y -207.201,Z 1718.671,A 0.000,B 0.000,C 90.000,E1 120.875} C_DIS
LIN {X -0.086,Y -209.546,Z 1718.665,A 0.000,B 0.000,C 90.000,E1 119.745} C_DIS
LIN {X -0.009,Y -333.806,Z 1718.665,A 0.000,B 0.000,C 90.000,E1 119.716} C_DIS
LIN {X -0.011,Y -340.052,Z 1718.664,A 0.000,B 0.000,C 90.000,E1 119.489} C_DIS
LIN {X -0.143,Y -342.881,Z 1718.663,A 0.000,B 0.000,C 90.000,E1 119.283} C_DIS
LIN {X -0.162,Y -346.611,Z 1718.660,A 0.000,B 0.000,C 90.000,E1 118.821} C_DIS
LIN {X 0.001,Y -348.324,Z 1718.658,A 0.000,B 0.000,C 90.000,E1 118.487} C_DIS
LIN {X 0.001,Y -362.708,Z 1718.641,A 0.000,B 0.000,C 90.000,E1 115.463} C_DIS
LIN {X -0.115,Y -377.233,Z 1718.627,A 0.000,B 0.000,C 90.000,E1 112.823} C_DIS
LIN {X 0.086,Y -391.528,Z 1718.614,A 0.000,B 0.000,C 90.000,E1 110.482} C_DIS
LIN {X 0.006,Y -407.229,Z 1718.601,A 0.000,B 0.000,C 90.000,E1 108.236} C_DIS
LIN {X 0.064,Y -424.443,Z 1718.589,A 0.000,B 0.000,C 90.000,E1 106.024} C_DIS
LIN {X 0.019,Y -443.291,Z 1718.577,A 0.000,B 0.000,C 90.000,E1 103.883} C_DIS
LIN {X -0.170,Y -463.236,Z 1718.566,A 0.000,B 0.000,C 90.000,E1 101.883} C_DIS
LIN {X -0.104,Y -486.313,Z 1718.554,A 0.000,B 0.000,C 90.000,E1 99.792} C_DIS
LIN {X -0.191,Y -507.244,Z 1718.545,A 0.000,B 0.000,C 90.000,E1 98.106} C_DIS
LIN {X 0.088,Y -509.213,Z 1718.544,A 0.000,B 0.000,C 90.000,E1 97.871} C_DIS
LIN {X -0.034,Y -510.979,Z 1718.542,A 0.000,B 0.000,C 90.000,E1 97.644} C_DIS
LIN {X -0.089,Y -512.299,Z 1718.541,A 0.000,B 0.000,C 90.000,E1 97.409} C_DIS
LIN {X 0.264,Y -513.922,Z 1718.538,A 0.000,B 0.000,C 90.000,E1 96.891} C_DIS
LIN {X 0.116,Y -514.442,Z 1718.536,A 0.000,B 0.000,C 90.000,E1 96.429} C_DIS
LIN {X -0.025,Y -513.945,Z 1718.533,A 0.000,B 0.000,C 90.000,E1 95.967} C_DIS
LIN {X -0.213,Y -512.346,Z 1718.531,A 0.000,B 0.000,C 90.000,E1 95.511} C_DIS
LIN {X 0.251,Y -511.041,Z 1718.529,A 0.000,B 0.000,C 90.000,E1 95.220} C_DIS
LIN {X -0.176,Y -502.063,Z 1718.522,A 0.000,B 0.000,C 90.000,E1 94.069} C_DIS
LIN {X -0.037,Y -489.437,Z 1718.513,A 0.000,B 0.000,C 90.000,E1 92.350} C_DIS
LIN {X 0.029,Y -478.506,Z 1718.505,A 0.000,B 0.000,C 90.000,E1 90.859} C_DIS
LIN {X 0.175,Y -465.747,Z 1718.495,A 0.000,B 0.000,C 90.000,E1 89.083} C_DIS
LIN {X -0.161,Y -451.015,Z 1718.484,A 0.000,B 0.000,C 90.000,E1 87.078} C_DIS
LIN {X 0.116,Y -436.227,Z 1718.472,A 0.000,B 0.000,C 90.000,E1 84.951} C_DIS
LIN {X -0.075,Y -423.330,Z 1718.462,A 0.000,B 0.000,C 90.000,E1 83.109} C_DIS
LIN {X -0.113,Y -405.461,Z 1718.447,A 0.000,B 0.000,C 90.000,E1 80.387} C_DIS
LIN {X -0.132,Y -388.639,Z 1718.431,A 0.000,B 0.000,C 90.000,E1 77.589} C_DIS
LIN {X -0.043,Y -375.752,Z 1718.418,A 0.000,B 0.000,C 90.000,E1 75.283} C_DIS
LIN {X -0.078,Y -361.726,Z 1718.404,A 0.000,B 0.000,C 90.000,E1 72.653} C_DIS
LIN {X -0.024,Y -346.631,Z 1718.387,A 0.000,B 0.000,C 90.000,E1 69.645} C_DIS
LIN {X 0.064,Y -336.519,Z 1718.375,A 0.000,B 0.000,C 90.000,E1 67.486} C_DIS
LIN {X 0.162,Y -325.055,Z 1718.361,A 0.000,B 0.000,C 90.000,E1 64.973} C_DIS
LIN {X -0.165,Y -314.038,Z 1718.347,A 0.000,B 0.000,C 90.000,E1 62.487} C_DIS
LIN {X -0.081,Y -304.480,Z 1718.334,A 0.000,B 0.000,C 90.000,E1 60.205} C_DIS
LIN {X 0.085,Y -294.964,Z 1718.322,A 0.000,B 0.000,C 90.000,E1 57.867} C_DIS
LIN {X -0.028,Y -286.726,Z 1718.310,A 0.000,B 0.000,C 90.000,E1 55.881} C_DIS
LIN {X -0.016,Y -276.999,Z 1718.297,A 0.000,B 0.000,C 90.000,E1 53.497} C_DIS
LIN {X -0.106,Y -267.129,Z 1718.284,A 0.000,B 0.000,C 90.000,E1 51.090} C_DIS
LIN {X -0.022,Y -256.054,Z 1718.268,A 0.000,B 0.000,C 90.000,E1 48.243} C_DIS
LIN {X 0.099,Y -245.301,Z 1718.252,A 0.000,B 0.000,C 90.000,E1 45.324} C_DIS
LIN {X 0.091,Y -233.912,Z 1718.233,A 0.000,B 0.000,C 90.000,E1 42.000} C_DIS
LIN {X 0.043,Y -224.536,Z 1718.217,A 0.000,B 0.000,C 90.000,E1 38.991} C_DIS
LIN {X -0.006,Y -216.055,Z 1718.200,A 0.000,B 0.000,C 90.000,E1 35.931} C_DIS
LIN {X 0.007,Y -208.354,Z 1718.182,A 0.000,B 0.000,C 90.000,E1 32.801} C_DIS
LIN {X 0.029,Y -201.458,Z 1718.165,A 0.000,B 0.000,C 90.000,E1 29.617} C_DIS
LIN {X -0.040,Y -195.146,Z 1718.147,A 0.000,B 0.000,C 90.000,E1 26.411} C_DIS
LIN {X -0.005,Y -189.435,Z 1718.129,A 0.000,B 0.000,C 90.000,E1 23.131} C_DIS
LIN {X 0.019,Y -184.324,Z 1718.110,A 0.000,B 0.000,C 90.000,E1 19.812} C_DIS
LIN {X 0.084,Y -180.024,Z 1718.091,A 0.000,B 0.000,C 90.000,E1 16.441} C_DIS
LIN {X -0.022,Y -175.635,Z 1718.068,A 0.000,B 0.000,C 90.000,E1 12.243} C_DIS
LIN {X -0.091,Y -172.231,Z 1718.044,A 0.000,B 0.000,C 90.000,E1 7.992} C_DIS
LIN {X -0.048,Y -169.463,Z 1718.016,A 0.000,B 0.000,C 90.000,E1 2.808} C_DIS
LIN {X 0.017,Y -168.127,Z 1717.969,A 0.000,B 0.000,C 90.000,E1 354.318} C_DIS
LIN {X -0.019,Y -169.695,Z 1717.925,A 0.000,B 0.000,C 90.000,E1 346.520} C_DIS
LIN {X -0.001,Y -172.317,Z 1717.896,A 0.000,B 0.000,C 90.000,E1 341.329} C_DIS
LIN {X -0.043,Y -175.620,Z 1717.872,A 0.000,B 0.000,C 90.000,E1 337.050} C_DIS
LIN {X -0.053,Y -179.855,Z 1717.849,A 0.000,B 0.000,C 90.000,E1 332.794} C_DIS
LIN {X -0.027,Y -184.064,Z 1717.830,A 0.000,B 0.000,C 90.000,E1 329.410} C_DIS
LIN {X -0.096,Y -189.233,Z 1717.811,A 0.000,B 0.000,C 90.000,E1 326.087} C_DIS
LIN {X 0.001,Y -193.790,Z 1717.798,A 0.000,B 0.000,C 90.000,E1 323.577} C_DIS
LIN {X 0.110,Y -199.087,Z 1717.784,A 0.000,B 0.000,C 90.000,E1 321.090} C_DIS
LIN {X -0.101,Y -206.118,Z 1717.768,A 0.000,B 0.000,C 90.000,E1 318.324} C_DIS
LIN {X 0.113,Y -214.184,Z 1717.753,A 0.000,B 0.000,C 90.000,E1 315.486} C_DIS
LIN {X -0.008,Y -221.925,Z 1717.740,A 0.000,B 0.000,C 90.000,E1 313.176} C_DIS
LIN {X 0.028,Y -230.601,Z 1717.727,A 0.000,B 0.000,C 90.000,E1 310.862} C_DIS
LIN {X -0.037,Y -238.697,Z 1717.717,A 0.000,B 0.000,C 90.000,E1 308.991} C_DIS
LIN {X -0.138,Y -247.792,Z 1717.706,A 0.000,B 0.000,C 90.000,E1 307.156} C_DIS
LIN {X -0.129,Y -262.245,Z 1717.692,A 0.000,B 0.000,C 90.000,E1 304.612} C_DIS
LIN {X 0.085,Y -280.595,Z 1717.677,A 0.000,B 0.000,C 90.000,E1 301.750} C_DIS
LIN {X 0.118,Y -302.770,Z 1717.660,A 0.000,B 0.000,C 90.000,E1 298.693} C_DIS
LIN {X 0.024,Y -318.180,Z 1717.649,A 0.000,B 0.000,C 90.000,E1 296.744} C_DIS
LIN {X 0.071,Y -333.848,Z 1717.638,A 0.000,B 0.000,C 90.000,E1 294.823} C_DIS
LIN {X 0.130,Y -346.795,Z 1717.629,A 0.000,B 0.000,C 90.000,E1 293.259} C_DIS
LIN {X -0.076,Y -359.507,Z 1717.621,A 0.000,B 0.000,C 90.000,E1 291.770} C_DIS
LIN {X -0.053,Y -371.495,Z 1717.613,A 0.000,B 0.000,C 90.000,E1 290.301} C_DIS
LIN {X 0.107,Y -378.356,Z 1717.608,A 0.000,B 0.000,C 90.000,E1 289.396} C_DIS
LIN {X -0.146,Y -382.459,Z 1717.605,A 0.000,B 0.000,C 90.000,E1 288.852} C_DIS
LIN {X 0.132,Y -387.863,Z 1717.600,A 0.000,B 0.000,C 90.000,E1 287.946} C_DIS
LIN {X 0.085,Y -392.283,Z 1717.595,A 0.000,B 0.000,C 90.000,E1 287.094} C_DIS
LIN {X -0.089,Y -394.696,Z 1717.592,A 0.000,B 0.000,C 90.000,E1 286.551} C_DIS
LIN {X 0.022,Y -396.732,Z 1717.589,A 0.000,B 0.000,C 90.000,E1 285.969} C_DIS
LIN {X -0.132,Y -398.390,Z 1717.586,A 0.000,B 0.000,C 90.000,E1 285.426} C_DIS
LIN {X 0.109,Y -399.734,Z 1717.583,A 0.000,B 0.000,C 90.000,E1 284.828} C_DIS
LIN {X -0.130,Y -400.671,Z 1717.579,A 0.000,B 0.000,C 90.000,E1 284.300} C_DIS
LIN {X 0.031,Y -401.252,Z 1717.576,A 0.000,B 0.000,C 90.000,E1 283.716} C_DIS
LIN {X -0.098,Y -401.384,Z 1717.573,A 0.000,B 0.000,C 90.000,E1 283.175} C_DIS
LIN {X 0.074,Y -401.163,Z 1717.570,A 0.000,B 0.000,C 90.000,E1 282.591} C_DIS
LIN {X -0.144,Y -400.443,Z 1717.567,A 0.000,B 0.000,C 90.000,E1 282.063} C_DIS
LIN {X 0.028,Y -399.243,Z 1717.564,A 0.000,B 0.000,C 90.000,E1 281.478} C_DIS
LIN {X 0.196,Y -397.575,Z 1717.561,A 0.000,B 0.000,C 90.000,E1 280.894} C_DIS
LIN {X -0.035,Y -395.350,Z 1717.558,A 0.000,B 0.000,C 90.000,E1 280.366} C_DIS
LIN {X 0.039,Y -392.499,Z 1717.554,A 0.000,B 0.000,C 90.000,E1 279.792} C_DIS
LIN {X -0.092,Y -382.279,Z 1717.545,A 0.000,B 0.000,C 90.000,E1 278.106} C_DIS
LIN {X -0.067,Y -376.985,Z 1717.540,A 0.000,B 0.000,C 90.000,E1 277.239} C_DIS
LIN {X -0.090,Y -372.927,Z 1717.537,A 0.000,B 0.000,C 90.000,E1 276.663} C_DIS
LIN {X -0.133,Y -368.310,Z 1717.534,A 0.000,B 0.000,C 90.000,E1 276.087} C_DIS
LIN {X 0.162,Y -363.017,Z 1717.530,A 0.000,B 0.000,C 90.000,E1 275.454} C_DIS
LIN {X -0.117,Y -357.236,Z 1717.527,A 0.000,B 0.000,C 90.000,E1 274.935} C_DIS
LIN {X -0.110,Y -351.191,Z 1717.524,A 0.000,B 0.000,C 90.000,E1 274.416} C_DIS
LIN {X 0.145,Y -344.927,Z 1717.522,A 0.000,B 0.000,C 90.000,E1 273.898} C_DIS
LIN {X -0.050,Y -338.502,Z 1717.519,A 0.000,B 0.000,C 90.000,E1 273.498} C_DIS
LIN {X 0.017,Y -332.016,Z 1717.517,A 0.000,B 0.000,C 90.000,E1 273.094} C_DIS
LIN {X -0.056,Y -325.441,Z 1717.515,A 0.000,B 0.000,C 90.000,E1 272.751} C_DIS
LIN {X 0.067,Y -318.732,Z 1717.513,A 0.000,B 0.000,C 90.000,E1 272.407} C_DIS
LIN {X -0.009,Y -307.994,Z 1717.511,A 0.000,B 0.000,C 90.000,E1 272.007} C_DIS
LIN {X 0.087,Y -297.624,Z 1717.509,A 0.000,B 0.000,C 90.000,E1 271.661} C_DIS
LIN {X 0.011,Y -290.467,Z 1717.508,A 0.000,B 0.000,C 90.000,E1 271.489} C_DIS
LIN {X -0.002,Y -278.555,Z 1717.507,A 0.000,B 0.000,C 90.000,E1 271.260} C_DIS
LIN {X -0.063,Y -265.622,Z 1717.506,A 0.000,B 0.000,C 90.000,E1 271.088} C_DIS
LIN {X -0.031,Y -255.976,Z 1717.505,A 0.000,B 0.000,C 90.000,E1 270.974} C_DIS
LIN {X -0.003,Y -243.951,Z 1717.505,A 0.000,B 0.000,C 90.000,E1 270.917} C_DIS
LIN {X -0.024,Y -181.477,Z 1717.505,A 0.000,B 0.000,C 90.000,E1 270.917} C_DIS
LIN {X 0.055,Y -181.563,Z 1717.500,A 0.000,B 0.000,C 90.000,E1 270.000} C_DIS
LIN {X 0.041,Y -180.853,Z 1717.472,A 0.000,B 0.000,C 90.000,E1 264.951} C_DIS
LIN {X -0.054,Y -178.964,Z 1717.444,A 0.000,B 0.000,C 90.000,E1 259.916} C_DIS
LIN {X -0.074,Y -177.914,Z 1717.434,A 0.000,B 0.000,C 90.000,E1 258.229} C_DIS
LIN {X -0.059,Y -175.549,Z 1717.411,A 0.000,B 0.000,C 90.000,E1 253.976} C_DIS
LIN {X -0.051,Y -172.281,Z 1717.387,A 0.000,B 0.000,C 90.000,E1 249.699} C_DIS
LIN {X -0.012,Y -171.760,Z 1717.382,A 0.000,B 0.000,C 90.000,E1 248.827} C_DIS
LIN {X 0.005,Y -167.360,Z 1717.354,A 0.000,B 0.000,C 90.000,E1 243.640} C_DIS
LIN {X 0.087,Y -166.748,Z 1717.349,A 0.000,B 0.000,C 90.000,E1 242.743} C_DIS
LIN {X -0.001,Y -162.729,Z 1717.324,A 0.000,B 0.000,C 90.000,E1 238.408} C_DIS
LIN {X 0.061,Y -161.419,Z 1717.315,A 0.000,B 0.000,C 90.000,E1 236.628} C_DIS
LIN {X 0.101,Y -157.412,Z 1717.290,A 0.000,B 0.000,C 90.000,E1 232.190} C_DIS
LIN {X 0.034,Y -155.413,Z 1717.275,A 0.000,B 0.000,C 90.000,E1 229.542} C_DIS
LIN {X -0.035,Y -151.741,Z 1717.250,A 0.000,B 0.000,C 90.000,E1 225.081} C_DIS
LIN {X -0.023,Y -149.938,Z 1717.235,A 0.000,B 0.000,C 90.000,E1 222.366} C_DIS
LIN {X 0.004,Y -146.786,Z 1717.210,A 0.000,B 0.000,C 90.000,E1 217.810} C_DIS
LIN {X -0.094,Y -145.359,Z 1717.195,A 0.000,B 0.000,C 90.000,E1 215.105} C_DIS
LIN {X 0.022,Y -142.428,Z 1717.164,A 0.000,B 0.000,C 90.000,E1 209.539} C_DIS
LIN {X 0.072,Y -141.417,Z 1717.149,A 0.000,B 0.000,C 90.000,E1 206.744} C_DIS
LIN {X 0.058,Y -139.361,Z 1717.113,A 0.000,B 0.000,C 90.000,E1 200.248} C_DIS
LIN {X 0.046,Y -138.804,Z 1717.097,A 0.000,B 0.000,C 90.000,E1 197.457} C_DIS
LIN {X -0.035,Y -138.349,Z 1717.056,A 0.000,B 0.000,C 90.000,E1 190.018} C_DIS
LIN {X -0.020,Y -139.364,Z 1717.009,A 0.000,B 0.000,C 90.000,E1 181.604} C_DIS
LIN {X 0.033,Y -141.250,Z 1716.973,A 0.000,B 0.000,C 90.000,E1 175.065} C_DIS
LIN {X -0.009,Y -142.618,Z 1716.957,A 0.000,B 0.000,C 90.000,E1 172.299} C_DIS
LIN {X -0.056,Y -144.936,Z 1716.932,A 0.000,B 0.000,C 90.000,E1 167.701} C_DIS
LIN {X 0.077,Y -147.565,Z 1716.911,A 0.000,B 0.000,C 90.000,E1 163.976} C_DIS
LIN {X -0.033,Y -150.173,Z 1716.891,A 0.000,B 0.000,C 90.000,E1 160.369} C_DIS
LIN {X -0.025,Y -153.547,Z 1716.871,A 0.000,B 0.000,C 90.000,E1 156.741} C_DIS
LIN {X 0.027,Y -156.965,Z 1716.851,A 0.000,B 0.000,C 90.000,E1 153.127} C_DIS
LIN {X -0.038,Y -161.073,Z 1716.831,A 0.000,B 0.000,C 90.000,E1 149.587} C_DIS
LIN {X 0.047,Y -163.180,Z 1716.821,A 0.000,B 0.000,C 90.000,E1 147.788} C_DIS
LIN {X 0.053,Y -167.602,Z 1716.802,A 0.000,B 0.000,C 90.000,E1 144.276} C_DIS
LIN {X -0.038,Y -171.430,Z 1716.787,A 0.000,B 0.000,C 90.000,E1 141.698} C_DIS
LIN {X 0.001,Y -176.350,Z 1716.768,A 0.000,B 0.000,C 90.000,E1 138.243} C_DIS
LIN {X -0.002,Y -180.641,Z 1716.754,A 0.000,B 0.000,C 90.000,E1 135.688} C_DIS
LIN {X -0.018,Y -186.043,Z 1716.735,A 0.000,B 0.000,C 90.000,E1 132.324} C_DIS
LIN {X 0.045,Y -190.678,Z 1716.721,A 0.000,B 0.000,C 90.000,E1 129.806} C_DIS
LIN {X 0.078,Y -196.430,Z 1716.703,A 0.000,B 0.000,C 90.000,E1 126.503} C_DIS
LIN {X 0.045,Y -201.215,Z 1716.689,A 0.000,B 0.000,C 90.000,E1 124.072} C_DIS
LIN {X -0.027,Y -207.169,Z 1716.672,A 0.000,B 0.000,C 90.000,E1 120.875} C_DIS
LIN {X 0.041,Y -209.472,Z 1716.665,A 0.000,B 0.000,C 90.000,E1 119.745} C_DIS
LIN {X 0.029,Y -333.071,Z 1716.665,A 0.000,B 0.000,C 90.000,E1 119.745} C_DIS
LIN {X -0.080,Y -334.717,Z 1716.665,A 0.000,B 0.000,C 90.000,E1 119.745} C_DIS
LIN {X 0.085,Y -340.115,Z 1716.664,A 0.000,B 0.000,C 90.000,E1 119.489} C_DIS
LIN {X -0.046,Y -342.872,Z 1716.663,A 0.000,B 0.000,C 90.000,E1 119.283} C_DIS
LIN {X -0.123,Y -346.605,Z 1716.660,A 0.000,B 0.000,C 90.000,E1 118.821} C_DIS
LIN {X 0.039,Y -348.284,Z 1716.658,A 0.000,B 0.000,C 90.000,E1 118.487} C_DIS
LIN {X -0.017,Y -361.138,Z 1716.643,A 0.000,B 0.000,C 90.000,E1 115.771} C_DIS
LIN {X 0.167,Y -375.480,Z 1716.628,A 0.000,B 0.000,C 90.000,E1 113.078} C_DIS
LIN {X -0.026,Y -389.602,Z 1716.615,A 0.000,B 0.000,C 90.000,E1 110.791} C_DIS
LIN {X -0.155,Y -405.118,Z 1716.603,A 0.000,B 0.000,C 90.000,E1 108.544} C_DIS
LIN {X -0.032,Y -422.132,Z 1716.591,A 0.000,B 0.000,C 90.000,E1 106.315} C_DIS
LIN {X -0.142,Y -440.763,Z 1716.579,A 0.000,B 0.000,C 90.000,E1 104.175} C_DIS
LIN {X -0.060,Y -460.622,Z 1716.567,A 0.000,B 0.000,C 90.000,E1 102.119} C_DIS
LIN {X -0.111,Y -483.653,Z 1716.556,A 0.000,B 0.000,C 90.000,E1 100.018} C_DIS
LIN {X -0.159,Y -507.141,Z 1716.545,A 0.000,B 0.000,C 90.000,E1 98.106} C_DIS
LIN {X 0.119,Y -509.079,Z 1716.544,A 0.000,B 0.000,C 90.000,E1 97.871} C_DIS
LIN {X -0.003,Y -510.819,Z 1716.542,A 0.000,B 0.000,C 90.000,E1 97.644} C_DIS
LIN {X -0.058,Y -512.120,Z 1716.541,A 0.000,B 0.000,C 90.000,E1 97.409} C_DIS
LIN {X -0.215,Y -513.713,Z 1716.538,A 0.000,B 0.000,C 90.000,E1 96.947} C_DIS
LIN {X 0.145,Y -514.209,Z 1716.536,A 0.000,B 0.000,C 90.000,E1 96.429} C_DIS
LIN {X 0.003,Y -513.687,Z 1716.533,A 0.000,B 0.000,C 90.000,E1 95.967} C_DIS
LIN {X -0.186,Y -512.058,Z 1716.531,A 0.000,B 0.000,C 90.000,E1 95.511} C_DIS
LIN {X -0.232,Y -510.735,Z 1716.529,A 0.000,B 0.000,C 90.000,E1 95.277} C_DIS
LIN {X 0.228,Y -499.965,Z 1716.521,A 0.000,B 0.000,C 90.000,E1 93.784} C_DIS
LIN {X -0.162,Y -487.307,Z 1716.512,A 0.000,B 0.000,C 90.000,E1 92.121} C_DIS
LIN {X 0.172,Y -474.581,Z 1716.502,A 0.000,B 0.000,C 90.000,E1 90.344} C_DIS
LIN {X -0.025,Y -463.591,Z 1716.494,A 0.000,B 0.000,C 90.000,E1 88.854} C_DIS
LIN {X -0.165,Y -450.702,Z 1716.484,A 0.000,B 0.000,C 90.000,E1 87.078} C_DIS
LIN {X 0.104,Y -435.900,Z 1716.472,A 0.000,B 0.000,C 90.000,E1 84.951} C_DIS
LIN {X 0.070,Y -421.162,Z 1716.460,A 0.000,B 0.000,C 90.000,E1 82.818} C_DIS
LIN {X -0.030,Y -403.379,Z 1716.445,A 0.000,B 0.000,C 90.000,E1 80.095} C_DIS
LIN {X -0.028,Y -386.626,Z 1716.429,A 0.000,B 0.000,C 90.000,E1 77.285} C_DIS
LIN {X -0.074,Y -373.749,Z 1716.417,A 0.000,B 0.000,C 90.000,E1 74.991} C_DIS
LIN {X 0.214,Y -361.295,Z 1716.404,A 0.000,B 0.000,C 90.000,E1 72.598} C_DIS
LIN {X 0.033,Y -346.191,Z 1716.387,A 0.000,B 0.000,C 90.000,E1 69.625} C_DIS
LIN {X -0.012,Y -334.597,Z 1716.373,A 0.000,B 0.000,C 90.000,E1 67.177} C_DIS
LIN {X 0.129,Y -321.826,Z 1716.358,A 0.000,B 0.000,C 90.000,E1 64.332} C_DIS
LIN {X 0.089,Y -312.201,Z 1716.345,A 0.000,B 0.000,C 90.000,E1 62.103} C_DIS
LIN {X -0.143,Y -302.677,Z 1716.333,A 0.000,B 0.000,C 90.000,E1 59.871} C_DIS
LIN {X -0.010,Y -293.185,Z 1716.320,A 0.000,B 0.000,C 90.000,E1 57.533} C_DIS
LIN {X 0.007,Y -284.922,Z 1716.308,A 0.000,B 0.000,C 90.000,E1 55.515} C_DIS
LIN {X -0.021,Y -275.161,Z 1716.295,A 0.000,B 0.000,C 90.000,E1 53.130} C_DIS
LIN {X -0.143,Y -265.312,Z 1716.282,A 0.000,B 0.000,C 90.000,E1 50.723} C_DIS
LIN {X 0.065,Y -254.264,Z 1716.266,A 0.000,B 0.000,C 90.000,E1 47.838} C_DIS
LIN {X -0.032,Y -243.570,Z 1716.250,A 0.000,B 0.000,C 90.000,E1 44.960} C_DIS
LIN {X 0.078,Y -232.304,Z 1716.231,A 0.000,B 0.000,C 90.000,E1 41.595} C_DIS
LIN {X 0.046,Y -224.191,Z 1716.216,A 0.000,B 0.000,C 90.000,E1 38.955} C_DIS
LIN {X 0.028,Y -215.770,Z 1716.199,A 0.000,B 0.000,C 90.000,E1 35.884} C_DIS
LIN {X 0.041,Y -208.099,Z 1716.182,A 0.000,B 0.000,C 90.000,E1 32.752} C_DIS
LIN {X -0.015,Y -201.263,Z 1716.164,A 0.000,B 0.000,C 90.000,E1 29.589} C_DIS
LIN {X -0.009,Y -194.966,Z 1716.146,A 0.000,B 0.000,C 90.000,E1 26.360} C_DIS
LIN {X 0.026,Y -189.284,Z 1716.128,A 0.000,B 0.000,C 90.000,E1 23.078} C_DIS
LIN {X 0.049,Y -184.189,Z 1716.110,A 0.000,B 0.000,C 90.000,E1 19.758} C_DIS
LIN {X -0.060,Y -179.903,Z 1716.091,A 0.000,B 0.000,C 90.000,E1 16.441} C_DIS
LIN {X 0.006,Y -175.522,Z 1716.068,A 0.000,B 0.000,C 90.000,E1 12.187} C_DIS
LIN {X -0.065,Y -172.123,Z 1716.044,A 0.000,B 0.000,C 90.000,E1 7.936} C_DIS
LIN {X -0.024,Y -169.379,Z 1716.015,A 0.000,B 0.000,C 90.000,E1 2.751} C_DIS
LIN {X 0.009,Y -168.090,Z 1715.964,A 0.000,B 0.000,C 90.000,E1 353.451} C_DIS
LIN {X 0.002,Y -169.979,Z 1715.920,A 0.000,B 0.000,C 90.000,E1 345.644} C_DIS
LIN {X -0.038,Y -172.836,Z 1715.891,A 0.000,B 0.000,C 90.000,E1 340.477} C_DIS
LIN {X 0.000,Y -176.358,Z 1715.868,A 0.000,B 0.000,C 90.000,E1 336.177} C_DIS
LIN {X 0.091,Y -180.786,Z 1715.844,A 0.000,B 0.000,C 90.000,E1 331.897} C_DIS
LIN {X 0.073,Y -185.268,Z 1715.825,A 0.000,B 0.000,C 90.000,E1 328.535} C_DIS
LIN {X -0.015,Y -190.719,Z 1715.807,A 0.000,B 0.000,C 90.000,E1 325.229} C_DIS
LIN {X -0.041,Y -195.527,Z 1715.793,A 0.000,B 0.000,C 90.000,E1 322.763} C_DIS
LIN {X -0.028,Y -202.104,Z 1715.777,A 0.000,B 0.000,C 90.000,E1 319.908} C_DIS
LIN {X 0.079,Y -208.457,Z 1715.764,A 0.000,B 0.000,C 90.000,E1 317.472} C_DIS
LIN {X -0.105,Y -216.825,Z 1715.749,A 0.000,B 0.000,C 90.000,E1 314.757} C_DIS
LIN {X -0.020,Y -224.901,Z 1715.736,A 0.000,B 0.000,C 90.000,E1 312.405} C_DIS
LIN {X 0.075,Y -233.946,Z 1715.723,A 0.000,B 0.000,C 90.000,E1 310.092} C_DIS
LIN {X -0.091,Y -242.430,Z 1715.712,A 0.000,B 0.000,C 90.000,E1 308.257} C_DIS
LIN {X 0.066,Y -249.989,Z 1715.704,A 0.000,B 0.000,C 90.000,E1 306.744} C_DIS
LIN {X 0.133,Y -264.654,Z 1715.690,A 0.000,B 0.000,C 90.000,E1 304.199} C_DIS
LIN {X 0.044,Y -283.152,Z 1715.675,A 0.000,B 0.000,C 90.000,E1 301.416} C_DIS
LIN {X -0.127,Y -302.929,Z 1715.660,A 0.000,B 0.000,C 90.000,E1 298.743} C_DIS
LIN {X 0.049,Y -318.309,Z 1715.649,A 0.000,B 0.000,C 90.000,E1 296.744} C_DIS
LIN {X -0.027,Y -333.927,Z 1715.638,A 0.000,B 0.000,C 90.000,E1 294.847} C_DIS
LIN {X 0.187,Y -346.802,Z 1715.629,A 0.000,B 0.000,C 90.000,E1 293.259} C_DIS
LIN {X -0.018,Y -359.548,Z 1715.621,A 0.000,B 0.000,C 90.000,E1 291.770} C_DIS
LIN {X -0.191,Y -369.314,Z 1715.614,A 0.000,B 0.000,C 90.000,E1 290.610} C_DIS
LIN {X -0.047,Y -376.321,Z 1715.609,A 0.000,B 0.000,C 90.000,E1 289.704} C_DIS
LIN {X 0.172,Y -380.642,Z 1715.606,A 0.000,B 0.000,C 90.000,E1 289.087} C_DIS
LIN {X 0.060,Y -386.325,Z 1715.601,A 0.000,B 0.000,C 90.000,E1 288.236} C_DIS
LIN {X -0.148,Y -389.629,Z 1715.598,A 0.000,B 0.000,C 90.000,E1 287.692} C_DIS
LIN {X 0.036,Y -392.498,Z 1715.595,A 0.000,B 0.000,C 90.000,E1 287.094} C_DIS
LIN {X -0.137,Y -394.890,Z 1715.592,A 0.000,B 0.000,C 90.000,E1 286.551} C_DIS
LIN {X -0.026,Y -396.923,Z 1715.589,A 0.000,B 0.000,C 90.000,E1 285.969} C_DIS
LIN {X -0.179,Y -398.608,Z 1715.586,A 0.000,B 0.000,C 90.000,E1 285.426} C_DIS
LIN {X 0.063,Y -399.941,Z 1715.582,A 0.000,B 0.000,C 90.000,E1 284.828} C_DIS
LIN {X -0.174,Y -400.875,Z 1715.579,A 0.000,B 0.000,C 90.000,E1 284.300} C_DIS
LIN {X -0.012,Y -401.452,Z 1715.576,A 0.000,B 0.000,C 90.000,E1 283.716} C_DIS
LIN {X -0.140,Y -401.598,Z 1715.573,A 0.000,B 0.000,C 90.000,E1 283.175} C_DIS
LIN {X 0.033,Y -401.381,Z 1715.570,A 0.000,B 0.000,C 90.000,E1 282.591} C_DIS
LIN {X -0.183,Y -400.665,Z 1715.567,A 0.000,B 0.000,C 90.000,E1 282.063} C_DIS
LIN {X -0.009,Y -399.481,Z 1715.564,A 0.000,B 0.000,C 90.000,E1 281.478} C_DIS
LIN {X 0.160,Y -397.787,Z 1715.561,A 0.000,B 0.000,C 90.000,E1 280.894} C_DIS
LIN {X -0.070,Y -395.514,Z 1715.557,A 0.000,B 0.000,C 90.000,E1 280.366} C_DIS
LIN {X 0.004,Y -392.680,Z 1715.554,A 0.000,B 0.000,C 90.000,E1 279.792} C_DIS
LIN {X -0.163,Y -384.101,Z 1715.547,A 0.000,B 0.000,C 90.000,E1 278.398} C_DIS
LIN {X -0.114,Y -378.916,Z 1715.542,A 0.000,B 0.000,C 90.000,E1 277.530} C_DIS
LIN {X -0.079,Y -375.100,Z 1715.539,A 0.000,B 0.000,C 90.000,E1 276.947} C_DIS
LIN {X -0.112,Y -370.764,Z 1715.535,A 0.000,B 0.000,C 90.000,E1 276.372} C_DIS
LIN {X -0.168,Y -365.826,Z 1715.532,A 0.000,B 0.000,C 90.000,E1 275.796} C_DIS
LIN {X 0.110,Y -360.050,Z 1715.529,A 0.000,B 0.000,C 90.000,E1 275.163} C_DIS
LIN {X 0.006,Y -354.209,Z 1715.526,A 0.000,B 0.000,C 90.000,E1 274.645} C_DIS
LIN {X -0.151,Y -348.188,Z 1715.523,A 0.000,B 0.000,C 90.000,E1 274.188} C_DIS
LIN {X -0.115,Y -341.769,Z 1715.521,A 0.000,B 0.000,C 90.000,E1 273.726} C_DIS
LIN {X 0.142,Y -335.186,Z 1715.518,A 0.000,B 0.000,C 90.000,E1 273.269} C_DIS
LIN {X 0.016,Y -325.368,Z 1715.515,A 0.000,B 0.000,C 90.000,E1 272.751} C_DIS
LIN {X -0.150,Y -318.652,Z 1715.514,A 0.000,B 0.000,C 90.000,E1 272.465} C_DIS
LIN {X -0.116,Y -311.626,Z 1715.512,A 0.000,B 0.000,C 90.000,E1 272.178} C_DIS
LIN {X -0.145,Y -301.198,Z 1715.510,A 0.000,B 0.000,C 90.000,E1 271.833} C_DIS
LIN {X 0.138,Y -290.581,Z 1715.508,A 0.000,B 0.000,C 90.000,E1 271.489} C_DIS
LIN {X 0.122,Y -278.890,Z 1715.507,A 0.000,B 0.000,C 90.000,E1 271.260} C_DIS
LIN {X 0.030,Y -265.776,Z 1715.506,A 0.000,B 0.000,C 90.000,E1 271.088} C_DIS
LIN {X 0.082,Y -256.287,Z 1715.505,A 0.000,B 0.000,C 90.000,E1 270.974} C_DIS
LIN {X 0.096,Y -242.919,Z 1715.505,A 0.000,B 0.000,C 90.000,E1 270.917} C_DIS
LIN {X 0.048,Y -181.471,Z 1715.505,A 0.000,B 0.000,C 90.000,E1 270.917} C_DIS
LIN {X -0.080,Y -181.546,Z 1715.500,A 0.000,B 0.000,C 90.000,E1 269.943} C_DIS
LIN {X 0.043,Y -180.908,Z 1715.475,A 0.000,B 0.000,C 90.000,E1 265.527} C_DIS
LIN {X -0.079,Y -180.767,Z 1715.471,A 0.000,B 0.000,C 90.000,E1 264.723} C_DIS
LIN {X -0.008,Y -178.861,Z 1715.442,A 0.000,B 0.000,C 90.000,E1 259.634} C_DIS
LIN {X 0.063,Y -175.904,Z 1715.414,A 0.000,B 0.000,C 90.000,E1 254.519} C_DIS
LIN {X 0.002,Y -174.585,Z 1715.405,A 0.000,B 0.000,C 90.000,E1 252.834} C_DIS
LIN {X 0.037,Y -171.569,Z 1715.381,A 0.000,B 0.000,C 90.000,E1 248.539} C_DIS
LIN {X 0.019,Y -167.792,Z 1715.357,A 0.000,B 0.000,C 90.000,E1 244.229} C_DIS
LIN {X 0.033,Y -166.508,Z 1715.347,A 0.000,B 0.000,C 90.000,E1 242.487} C_DIS
LIN {X 0.029,Y -163.216,Z 1715.328,A 0.000,B 0.000,C 90.000,E1 238.997} C_DIS
LIN {X -0.007,Y -161.182,Z 1715.313,A 0.000,B 0.000,C 90.000,E1 236.373} C_DIS
LIN {X -0.006,Y -157.195,Z 1715.289,A 0.000,B 0.000,C 90.000,E1 231.949} C_DIS
LIN {X 0.039,Y -155.924,Z 1715.279,A 0.000,B 0.000,C 90.000,E1 230.150} C_DIS
LIN {X -0.011,Y -152.175,Z 1715.254,A 0.000,B 0.000,C 90.000,E1 225.688} C_DIS
LIN {X 0.005,Y -150.423,Z 1715.239,A 0.000,B 0.000,C 90.000,E1 222.975} C_DIS
LIN {X -0.070,Y -147.151,Z 1715.214,A 0.000,B 0.000,C 90.000,E1 218.463} C_DIS
LIN {X 0.018,Y -145.164,Z 1715.193,A 0.000,B 0.000,C 90.000,E1 214.771} C_DIS
LIN {X -0.066,Y -142.318,Z 1715.162,A 0.000,B 0.000,C 90.000,E1 209.283} C_DIS
LIN {X 0.054,Y -141.707,Z 1715.152,A 0.000,B 0.000,C 90.000,E1 207.385} C_DIS
LIN {X -0.023,Y -139.470,Z 1715.116,A 0.000,B 0.000,C 90.000,E1 200.918} C_DIS
LIN {X 0.031,Y -139.202,Z 1715.106,A 0.000,B 0.000,C 90.000,E1 199.033} C_DIS
LIN {X -0.042,Y -138.328,Z 1715.054,A 0.000,B 0.000,C 90.000,E1 189.726} C_DIS
LIN {X -0.040,Y -139.442,Z 1715.007,A 0.000,B 0.000,C 90.000,E1 181.318} C_DIS
LIN {X 0.040,Y -140.976,Z 1714.976,A 0.000,B 0.000,C 90.000,E1 175.698} C_DIS
LIN {X -0.010,Y -142.732,Z 1714.956,A 0.000,B 0.000,C 90.000,E1 172.008} C_DIS
LIN {X -0.053,Y -145.120,Z 1714.930,A 0.000,B 0.000,C 90.000,E1 167.409} C_DIS
LIN {X -0.059,Y -147.744,Z 1714.910,A 0.000,B 0.000,C 90.000,E1 163.740} C_DIS
LIN {X 0.022,Y -150.411,Z 1714.889,A 0.000,B 0.000,C 90.000,E1 160.061} C_DIS
LIN {X 0.038,Y -153.849,Z 1714.869,A 0.000,B 0.000,C 90.000,E1 156.433} C_DIS
LIN {X -0.044,Y -157.259,Z 1714.849,A 0.000,B 0.000,C 90.000,E1 152.871} C_DIS
LIN {X 0.034,Y -161.434,Z 1714.829,A 0.000,B 0.000,C 90.000,E1 149.282} C_DIS
LIN {X 0.041,Y -165.635,Z 1714.810,A 0.000,B 0.000,C 90.000,E1 145.754} C_DIS
LIN {X 0.023,Y -170.567,Z 1714.790,A 0.000,B 0.000,C 90.000,E1 142.271} C_DIS
LIN {X -0.069,Y -175.444,Z 1714.771,A 0.000,B 0.000,C 90.000,E1 138.852} C_DIS
LIN {X 0.047,Y -181.067,Z 1714.752,A 0.000,B 0.000,C 90.000,E1 135.405} C_DIS
LIN {X 0.037,Y -186.505,Z 1714.734,A 0.000,B 0.000,C 90.000,E1 132.043} C_DIS
LIN {X -0.021,Y -191.125,Z 1714.720,A 0.000,B 0.000,C 90.000,E1 129.564} C_DIS
LIN {X -0.101,Y -196.922,Z 1714.702,A 0.000,B 0.000,C 90.000,E1 126.297} C_DIS
LIN {X 0.095,Y -200.185,Z 1714.692,A 0.000,B 0.000,C 90.000,E1 124.612} C_DIS
LIN {X 0.091,Y -207.680,Z 1714.670,A 0.000,B 0.000,C 90.000,E1 120.590} C_DIS
LIN {X -0.033,Y -209.409,Z 1714.666,A 0.000,B 0.000,C 90.000,E1 119.795} C_DIS
LIN {X -0.104,Y -333.519,Z 1714.665,A 0.000,B 0.000,C 90.000,E1 119.795} C_DIS
LIN {X 0.084,Y -334.718,Z 1714.665,A 0.000,B 0.000,C 90.000,E1 119.745} C_DIS
LIN {X -0.077,Y -339.314,Z 1714.664,A 0.000,B 0.000,C 90.000,E1 119.589} C_DIS
LIN {X -0.113,Y -341.794,Z 1714.663,A 0.000,B 0.000,C 90.000,E1 119.411} C_DIS
LIN {X -0.012,Y -345.139,Z 1714.661,A 0.000,B 0.000,C 90.000,E1 119.027} C_DIS
LIN {X -0.071,Y -347.042,Z 1714.660,A 0.000,B 0.000,C 90.000,E1 118.743} C_DIS
LIN {X -0.125,Y -349.882,Z 1714.656,A 0.000,B 0.000,C 90.000,E1 118.153} C_DIS
LIN {X 0.031,Y -362.903,Z 1714.641,A 0.000,B 0.000,C 90.000,E1 115.412} C_DIS
LIN {X -0.067,Y -377.452,Z 1714.626,A 0.000,B 0.000,C 90.000,E1 112.770} C_DIS
LIN {X 0.147,Y -391.773,Z 1714.614,A 0.000,B 0.000,C 90.000,E1 110.429} C_DIS
LIN {X 0.082,Y -407.500,Z 1714.601,A 0.000,B 0.000,C 90.000,E1 108.181} C_DIS
LIN {X 0.155,Y -424.744,Z 1714.589,A 0.000,B 0.000,C 90.000,E1 105.969} C_DIS
LIN {X 0.135,Y -443.614,Z 1714.577,A 0.000,B 0.000,C 90.000,E1 103.828} C_DIS
LIN {X -0.021,Y -463.570,Z 1714.566,A 0.000,B 0.000,C 90.000,E1 101.827} C_DIS
LIN {X 0.146,Y -486.687,Z 1714.554,A 0.000,B 0.000,C 90.000,E1 99.726} C_DIS
LIN {X -0.181,Y -505.061,Z 1714.546,A 0.000,B 0.000,C 90.000,E1 98.276} C_DIS
LIN {X 0.009,Y -507.465,Z 1714.545,A 0.000,B 0.000,C 90.000,E1 98.049} C_DIS
LIN {X 0.241,Y -510.855,Z 1714.542,A 0.000,B 0.000,C 90.000,E1 97.587} C_DIS
LIN {X 0.187,Y -512.084,Z 1714.541,A 0.000,B 0.000,C 90.000,E1 97.352} C_DIS
LIN {X 0.068,Y -512.975,Z 1714.540,A 0.000,B 0.000,C 90.000,E1 97.125} C_DIS
LIN {X -0.079,Y -513.896,Z 1714.537,A 0.000,B 0.000,C 90.000,E1 96.663} C_DIS
LIN {X -0.223,Y -513.789,Z 1714.534,A 0.000,B 0.000,C 90.000,E1 96.201} C_DIS
LIN {X 0.149,Y -512.633,Z 1714.532,A 0.000,B 0.000,C 90.000,E1 95.682} C_DIS
LIN {X 0.055,Y -511.606,Z 1714.530,A 0.000,B 0.000,C 90.000,E1 95.454} C_DIS
LIN {X 0.008,Y -510.209,Z 1714.529,A 0.000,B 0.000,C 90.000,E1 95.220} C_DIS
LIN {X 0.210,Y -495.808,Z 1714.518,A 0.000,B 0.000,C 90.000,E1 93.269} C_DIS
LIN {X 0.086,Y -481.337,Z 1714.507,A 0.000,B 0.000,C 90.000,E1 91.318} C_DIS
LIN {X -0.187,Y -468.561,Z 1714.498,A 0.000,B 0.000,C 90.000,E1 89.599} C_DIS
LIN {X -0.221,Y -455.663,Z 1714.488,A 0.000,B 0.000,C 90.000,E1 87.822} C_DIS
LIN {X 0.183,Y -444.549,Z 1714.479,A 0.000,B 0.000,C 90.000,E1 86.216} C_DIS
LIN {X 0.155,Y -431.618,Z 1714.469,A 0.000,B 0.000,C 90.000,E1 84.375} C_DIS
LIN {X 0.163,Y -415.130,Z 1714.455,A 0.000,B 0.000,C 90.000,E1 81.951} C_DIS
LIN {X 0.036,Y -395.942,Z 1714.438,A 0.000,B 0.000,C 90.000,E1 78.926} C_DIS
LIN {X 0.162,Y -381.144,Z 1714.424,A 0.000,B 0.000,C 90.000,E1 76.353} C_DIS
LIN {X 0.147,Y -366.855,Z 1714.410,A 0.000,B 0.000,C 90.000,E1 73.740} C_DIS
LIN {X -0.081,Y -354.509,Z 1714.397,A 0.000,B 0.000,C 90.000,E1 71.402} C_DIS
LIN {X 0.102,Y -339.712,Z 1714.380,A 0.000,B 0.000,C 90.000,E1 68.337} C_DIS
LIN {X 0.019,Y -328.201,Z 1714.366,A 0.000,B 0.000,C 90.000,E1 65.869} C_DIS
LIN {X 0.124,Y -315.701,Z 1714.350,A 0.000,B 0.000,C 90.000,E1 62.999} C_DIS
LIN {X -0.137,Y -304.780,Z 1714.336,A 0.000,B 0.000,C 90.000,E1 60.461} C_DIS
LIN {X 0.052,Y -293.948,Z 1714.321,A 0.000,B 0.000,C 90.000,E1 57.788} C_DIS
LIN {X -0.060,Y -287.097,Z 1714.312,A 0.000,B 0.000,C 90.000,E1 56.135} C_DIS
LIN {X -0.030,Y -277.374,Z 1714.299,A 0.000,B 0.000,C 90.000,E1 53.749} C_DIS
LIN {X -0.061,Y -267.502,Z 1714.285,A 0.000,B 0.000,C 90.000,E1 51.331} C_DIS
LIN {X 0.025,Y -256.358,Z 1714.269,A 0.000,B 0.000,C 90.000,E1 48.485} C_DIS
LIN {X -0.022,Y -246.917,Z 1714.255,A 0.000,B 0.000,C 90.000,E1 45.972} C_DIS
LIN {X 0.043,Y -236.635,Z 1714.239,A 0.000,B 0.000,C 90.000,E1 43.014} C_DIS
LIN {X -0.014,Y -225.918,Z 1714.220,A 0.000,B 0.000,C 90.000,E1 39.644} C_DIS
LIN {X 0.069,Y -216.363,Z 1714.201,A 0.000,B 0.000,C 90.000,E1 36.171} C_DIS
LIN {X -0.078,Y -208.638,Z 1714.184,A 0.000,B 0.000,C 90.000,E1 33.086} C_DIS
LIN {X 0.058,Y -201.768,Z 1714.166,A 0.000,B 0.000,C 90.000,E1 29.873} C_DIS
LIN {X -0.005,Y -195.433,Z 1714.148,A 0.000,B 0.000,C 90.000,E1 26.668} C_DIS
LIN {X -0.048,Y -188.363,Z 1714.125,A 0.000,B 0.000,C 90.000,E1 22.589} C_DIS
LIN {X -0.045,Y -183.393,Z 1714.107,A 0.000,B 0.000,C 90.000,E1 19.268} C_DIS
LIN {X -0.002,Y -179.243,Z 1714.088,A 0.000,B 0.000,C 90.000,E1 15.898} C_DIS
LIN {X -0.001,Y -174.986,Z 1714.065,A 0.000,B 0.000,C 90.000,E1 11.658} C_DIS
LIN {X 0.077,Y -171.699,Z 1714.041,A 0.000,B 0.000,C 90.000,E1 7.352} C_DIS
LIN {X 0.070,Y -169.125,Z 1714.012,A 0.000,B 0.000,C 90.000,E1 2.178} C_DIS
LIN {X 0.006,Y -168.019,Z 1713.964,A 0.000,B 0.000,C 90.000,E1 353.451} C_DIS
LIN {X -0.004,Y -169.910,Z 1713.920,A 0.000,B 0.000,C 90.000,E1 345.644} C_DIS
LIN {X -0.047,Y -172.787,Z 1713.891,A 0.000,B 0.000,C 90.000,E1 340.477} C_DIS
LIN {X -0.011,Y -176.309,Z 1713.868,A 0.000,B 0.000,C 90.000,E1 336.177} C_DIS
LIN {X 0.079,Y -180.754,Z 1713.844,A 0.000,B 0.000,C 90.000,E1 331.897} C_DIS
LIN {X 0.059,Y -185.262,Z 1713.825,A 0.000,B 0.000,C 90.000,E1 328.535} C_DIS
LIN {X -0.028,Y -190.746,Z 1713.807,A 0.000,B 0.000,C 90.000,E1 325.229} C_DIS
LIN {X -0.055,Y -195.601,Z 1713.793,A 0.000,B 0.000,C 90.000,E1 322.763} C_DIS
LIN {X -0.040,Y -202.203,Z 1713.777,A 0.000,B 0.000,C 90.000,E1 319.908} C_DIS
LIN {X 0.068,Y -208.588,Z 1713.764,A 0.000,B 0.000,C 90.000,E1 317.472} C_DIS
LIN {X -0.113,Y -216.981,Z 1713.749,A 0.000,B 0.000,C 90.000,E1 314.757} C_DIS
LIN {X -0.026,Y -225.096,Z 1713.736,A 0.000,B 0.000,C 90.000,E1 312.405} C_DIS
LIN {X 0.075,Y -234.169,Z 1713.723,A 0.000,B 0.000,C 90.000,E1 310.092} C_DIS
LIN {X -0.088,Y -242.669,Z 1713.712,A 0.000,B 0.000,C 90.000,E1 308.257} C_DIS
LIN {X 0.072,Y -250.231,Z 1713.704,A 0.000,B 0.000,C 90.000,E1 306.744} C_DIS
LIN {X -0.110,Y -262.669,Z 1713.692,A 0.000,B 0.000,C 90.000,E1 304.612} C_DIS
LIN {X -0.123,Y -280.940,Z 1713.677,A 0.000,B 0.000,C 90.000,E1 301.799} C_DIS
LIN {X -0.104,Y -300.555,Z 1713.661,A 0.000,B 0.000,C 90.000,E1 299.077} C_DIS
LIN {X 0.027,Y -315.845,Z 1713.651,A 0.000,B 0.000,C 90.000,E1 297.078} C_DIS
LIN {X 0.038,Y -331.424,Z 1713.640,A 0.000,B 0.000,C 90.000,E1 295.155} C_DIS
LIN {X 0.057,Y -344.348,Z 1713.631,A 0.000,B 0.000,C 90.000,E1 293.590} C_DIS
LIN {X -0.001,Y -359.630,Z 1713.621,A 0.000,B 0.000,C 90.000,E1 291.770} C_DIS
LIN {X -0.144,Y -371.862,Z 1713.613,A 0.000,B 0.000,C 90.000,E1 290.301} C_DIS
LIN {X 0.018,Y -378.717,Z 1713.608,A 0.000,B 0.000,C 90.000,E1 289.396} C_DIS
LIN {X -0.104,Y -384.690,Z 1713.603,A 0.000,B 0.000,C 90.000,E1 288.544} C_DIS
LIN {X 0.046,Y -388.216,Z 1713.600,A 0.000,B 0.000,C 90.000,E1 287.946} C_DIS
LIN {X -0.151,Y -391.289,Z 1713.597,A 0.000,B 0.000,C 90.000,E1 287.402} C_DIS
LIN {X 0.208,Y -395.100,Z 1713.592,A 0.000,B 0.000,C 90.000,E1 286.496} C_DIS
LIN {X -0.059,Y -397.123,Z 1713.589,A 0.000,B 0.000,C 90.000,E1 285.969} C_DIS
LIN {X 0.175,Y -398.804,Z 1713.586,A 0.000,B 0.000,C 90.000,E1 285.371} C_DIS
LIN {X 0.032,Y -400.137,Z 1713.582,A 0.000,B 0.000,C 90.000,E1 284.828} C_DIS
LIN {X -0.203,Y -401.071,Z 1713.579,A 0.000,B 0.000,C 90.000,E1 284.300} C_DIS
LIN {X 0.055,Y -401.653,Z 1713.576,A 0.000,B 0.000,C 90.000,E1 283.703} C_DIS
LIN {X -0.167,Y -401.838,Z 1713.573,A 0.000,B 0.000,C 90.000,E1 283.175} C_DIS
LIN {X 0.008,Y -401.559,Z 1713.570,A 0.000,B 0.000,C 90.000,E1 282.591} C_DIS
LIN {X 0.184,Y -400.878,Z 1713.567,A 0.000,B 0.000,C 90.000,E1 282.007} C_DIS
LIN {X -0.033,Y -399.678,Z 1713.564,A 0.000,B 0.000,C 90.000,E1 281.478} C_DIS
LIN {X 0.138,Y -397.965,Z 1713.561,A 0.000,B 0.000,C 90.000,E1 280.894} C_DIS
LIN {X -0.091,Y -395.704,Z 1713.557,A 0.000,B 0.000,C 90.000,E1 280.366} C_DIS
LIN {X -0.014,Y -392.864,Z 1713.554,A 0.000,B 0.000,C 90.000,E1 279.792} C_DIS
LIN {X -0.165,Y -386.060,Z 1713.548,A 0.000,B 0.000,C 90.000,E1 278.681} C_DIS
LIN {X -0.128,Y -379.054,Z 1713.542,A 0.000,B 0.000,C 90.000,E1 277.530} C_DIS
LIN {X -0.130,Y -373.080,Z 1713.537,A 0.000,B 0.000,C 90.000,E1 276.663} C_DIS
LIN {X -0.172,Y -368.440,Z 1713.534,A 0.000,B 0.000,C 90.000,E1 276.087} C_DIS
LIN {X 0.128,Y -363.059,Z 1713.530,A 0.000,B 0.000,C 90.000,E1 275.454} C_DIS
LIN {X -0.152,Y -357.198,Z 1713.527,A 0.000,B 0.000,C 90.000,E1 274.935} C_DIS
LIN {X -0.137,Y -351.103,Z 1713.524,A 0.000,B 0.000,C 90.000,E1 274.416} C_DIS
LIN {X 0.157,Y -344.773,Z 1713.522,A 0.000,B 0.000,C 90.000,E1 273.898} C_DIS
LIN {X -0.003,Y -338.334,Z 1713.519,A 0.000,B 0.000,C 90.000,E1 273.498} C_DIS
LIN {X 0.081,Y -331.725,Z 1713.517,A 0.000,B 0.000,C 90.000,E1 273.094} C_DIS
LIN {X 0.056,Y -325.161,Z 1713.515,A 0.000,B 0.000,C 90.000,E1 272.751} C_DIS
LIN {X 0.076,Y -315.012,Z 1713.513,A 0.000,B 0.000,C 90.000,E1 272.293} C_DIS
LIN {X -0.076,Y -304.583,Z 1713.511,A 0.000,B 0.000,C 90.000,E1 271.949} C_DIS
LIN {X 0.108,Y -293.978,Z 1713.509,A 0.000,B 0.000,C 90.000,E1 271.604} C_DIS
LIN {X 0.000,Y -282.645,Z 1713.508,A 0.000,B 0.000,C 90.000,E1 271.375} C_DIS
LIN {X 0.134,Y -270.453,Z 1713.506,A 0.000,B 0.000,C 90.000,E1 271.146} C_DIS
LIN {X -0.071,Y -256.552,Z 1713.506,A 0.000,B 0.000,C 90.000,E1 271.031} C_DIS
LIN {X -0.018,Y -246.554,Z 1713.505,A 0.000,B 0.000,C 90.000,E1 270.974} C_DIS
LIN {X -0.036,Y -181.465,Z 1713.505,A 0.000,B 0.000,C 90.000,E1 270.974} C_DIS
LIN {X 0.015,Y -181.552,Z 1713.500,A 0.000,B 0.000,C 90.000,E1 269.943} C_DIS
LIN {X -0.042,Y -180.908,Z 1713.475,A 0.000,B 0.000,C 90.000,E1 265.584} C_DIS
LIN {X 0.016,Y -180.779,Z 1713.471,A 0.000,B 0.000,C 90.000,E1 264.723} C_DIS
LIN {X -0.090,Y -178.874,Z 1713.443,A 0.000,B 0.000,C 90.000,E1 259.690} C_DIS
LIN {X -0.013,Y -175.917,Z 1713.414,A 0.000,B 0.000,C 90.000,E1 254.574} C_DIS
LIN {X 0.044,Y -174.611,Z 1713.405,A 0.000,B 0.000,C 90.000,E1 252.851} C_DIS
LIN {X -0.030,Y -171.593,Z 1713.381,A 0.000,B 0.000,C 90.000,E1 248.592} C_DIS
LIN {X -0.042,Y -167.815,Z 1713.357,A 0.000,B 0.000,C 90.000,E1 244.280} C_DIS
LIN {X -0.024,Y -166.537,Z 1713.347,A 0.000,B 0.000,C 90.000,E1 242.538} C_DIS
LIN {X 0.025,Y -162.535,Z 1713.323,A 0.000,B 0.000,C 90.000,E1 238.152} C_DIS
LIN {X -0.053,Y -161.211,Z 1713.313,A 0.000,B 0.000,C 90.000,E1 236.421} C_DIS
LIN {X -0.017,Y -157.219,Z 1713.289,A 0.000,B 0.000,C 90.000,E1 231.984} C_DIS
LIN {X 0.006,Y -155.945,Z 1713.279,A 0.000,B 0.000,C 90.000,E1 230.194} C_DIS
LIN {X -0.034,Y -152.198,Z 1713.254,A 0.000,B 0.000,C 90.000,E1 225.729} C_DIS
LIN {X -0.014,Y -150.444,Z 1713.239,A 0.000,B 0.000,C 90.000,E1 223.014} C_DIS
LIN {X 0.014,Y -147.170,Z 1713.214,A 0.000,B 0.000,C 90.000,E1 218.463} C_DIS
LIN {X -0.019,Y -145.186,Z 1713.193,A 0.000,B 0.000,C 90.000,E1 214.818} C_DIS
LIN {X 0.015,Y -142.330,Z 1713.163,A 0.000,B 0.000,C 90.000,E1 209.283} C_DIS
LIN {X -0.055,Y -141.719,Z 1713.152,A 0.000,B 0.000,C 90.000,E1 207.462} C_DIS
LIN {X 0.058,Y -139.476,Z 1713.116,A 0.000,B 0.000,C 90.000,E1 200.918} C_DIS
LIN {X 0.049,Y -138.972,Z 1713.101,A 0.000,B 0.000,C 90.000,E1 198.127} C_DIS
LIN {X 0.038,Y -138.331,Z 1713.054,A 0.000,B 0.000,C 90.000,E1 189.726} C_DIS
LIN {X 0.041,Y -139.435,Z 1713.007,A 0.000,B 0.000,C 90.000,E1 181.318} C_DIS
LIN {X -0.019,Y -140.963,Z 1712.976,A 0.000,B 0.000,C 90.000,E1 175.755} C_DIS
LIN {X 0.072,Y -142.719,Z 1712.956,A 0.000,B 0.000,C 90.000,E1 172.008} C_DIS
LIN {X 0.030,Y -145.099,Z 1712.930,A 0.000,B 0.000,C 90.000,E1 167.409} C_DIS
LIN {X 0.026,Y -147.724,Z 1712.910,A 0.000,B 0.000,C 90.000,E1 163.740} C_DIS
LIN {X -0.033,Y -150.383,Z 1712.889,A 0.000,B 0.000,C 90.000,E1 160.115} C_DIS
LIN {X -0.016,Y -153.814,Z 1712.869,A 0.000,B 0.000,C 90.000,E1 156.485} C_DIS
LIN {X 0.043,Y -157.226,Z 1712.849,A 0.000,B 0.000,C 90.000,E1 152.871} C_DIS
LIN {X -0.016,Y -161.394,Z 1712.830,A 0.000,B 0.000,C 90.000,E1 149.331} C_DIS
LIN {X -0.006,Y -165.595,Z 1712.810,A 0.000,B 0.000,C 90.000,E1 145.801} C_DIS
LIN {X -0.020,Y -170.518,Z 1712.791,A 0.000,B 0.000,C 90.000,E1 142.316} C_DIS
LIN {X 0.024,Y -175.398,Z 1712.771,A 0.000,B 0.000,C 90.000,E1 138.852} C_DIS
LIN {X 0.016,Y -181.022,Z 1712.752,A 0.000,B 0.000,C 90.000,E1 135.445} C_DIS
LIN {X 0.009,Y -186.453,Z 1712.734,A 0.000,B 0.000,C 90.000,E1 132.081} C_DIS
LIN {X 0.079,Y -191.077,Z 1712.720,A 0.000,B 0.000,C 90.000,E1 129.564} C_DIS
LIN {X 0.000,Y -196.866,Z 1712.702,A 0.000,B 0.000,C 90.000,E1 126.297} C_DIS
LIN {X -0.082,Y -200.125,Z 1712.693,A 0.000,B 0.000,C 90.000,E1 124.692} C_DIS
LIN {X -0.091,Y -207.622,Z 1712.670,A 0.000,B 0.000,C 90.000,E1 120.669} C_DIS
LIN {X 0.103,Y -209.330,Z 1712.666,A 0.000,B 0.000,C 90.000,E1 119.795} C_DIS
LIN {X 0.112,Y -332.936,Z 1712.666,A 0.000,B 0.000,C 90.000,E1 119.795} C_DIS
LIN {X -0.040,Y -334.805,Z 1712.666,A 0.000,B 0.000,C 90.000,E1 119.795} C_DIS
LIN {X -0.077,Y -339.222,Z 1712.664,A 0.000,B 0.000,C 90.000,E1 119.617} C_DIS
LIN {X 0.057,Y -341.675,Z 1712.663,A 0.000,B 0.000,C 90.000,E1 119.411} C_DIS
LIN {X -0.144,Y -345.001,Z 1712.661,A 0.000,B 0.000,C 90.000,E1 119.077} C_DIS
LIN {X 0.092,Y -346.906,Z 1712.660,A 0.000,B 0.000,C 90.000,E1 118.743} C_DIS
LIN {X 0.033,Y -349.745,Z 1712.656,A 0.000,B 0.000,C 90.000,E1 118.153} C_DIS
LIN {X -0.137,Y -362.751,Z 1712.641,A 0.000,B 0.000,C 90.000,E1 115.463} C_DIS
LIN {X 0.095,Y -377.284,Z 1712.627,A 0.000,B 0.000,C 90.000,E1 112.770} C_DIS
LIN {X -0.057,Y -391.590,Z 1712.614,A 0.000,B 0.000,C 90.000,E1 110.482} C_DIS
LIN {X -0.140,Y -407.303,Z 1712.601,A 0.000,B 0.000,C 90.000,E1 108.236} C_DIS
LIN {X -0.086,Y -424.531,Z 1712.589,A 0.000,B 0.000,C 90.000,E1 106.024} C_DIS
LIN {X -0.127,Y -443.383,Z 1712.577,A 0.000,B 0.000,C 90.000,E1 103.883} C_DIS
LIN {X 0.140,Y -463.334,Z 1712.566,A 0.000,B 0.000,C 90.000,E1 101.827} C_DIS
LIN {X -0.181,Y -486.444,Z 1712.554,A 0.000,B 0.000,C 90.000,E1 99.782} C_DIS
LIN {X -0.034,Y -504.815,Z 1712.546,A 0.000,B 0.000,C 90.000,E1 98.276} C_DIS
LIN {X 0.155,Y -507.222,Z 1712.545,A 0.000,B 0.000,C 90.000,E1 98.049} C_DIS
LIN {X -0.118,Y -510.613,Z 1712.542,A 0.000,B 0.000,C 90.000,E1 97.644} C_DIS
LIN {X -0.173,Y -511.842,Z 1712.541,A 0.000,B 0.000,C 90.000,E1 97.409} C_DIS
LIN {X 0.215,Y -512.734,Z 1712.540,A 0.000,B 0.000,C 90.000,E1 97.125} C_DIS
LIN {X 0.066,Y -513.655,Z 1712.537,A 0.000,B 0.000,C 90.000,E1 96.663} C_DIS
LIN {X -0.079,Y -513.550,Z 1712.534,A 0.000,B 0.000,C 90.000,E1 96.201} C_DIS
LIN {X -0.218,Y -512.398,Z 1712.532,A 0.000,B 0.000,C 90.000,E1 95.739} C_DIS
LIN {X 0.195,Y -511.372,Z 1712.530,A 0.000,B 0.000,C 90.000,E1 95.454} C_DIS
LIN {X 0.149,Y -509.976,Z 1712.529,A 0.000,B 0.000,C 90.000,E1 95.220} C_DIS
LIN {X -0.154,Y -495.598,Z 1712.518,A 0.000,B 0.000,C 90.000,E1 93.326} C_DIS
LIN {X 0.210,Y -481.140,Z 1712.507,A 0.000,B 0.000,C 90.000,E1 91.318} C_DIS
LIN {X -0.071,Y -468.375,Z 1712.498,A 0.000,B 0.000,C 90.000,E1 89.599} C_DIS
LIN {X -0.112,Y -455.471,Z 1712.488,A 0.000,B 0.000,C 90.000,E1 87.822} C_DIS
LIN {X -0.157,Y -444.341,Z 1712.479,A 0.000,B 0.000,C 90.000,E1 86.274} C_DIS
LIN {X -0.179,Y -431.383,Z 1712.469,A 0.000,B 0.000,C 90.000,E1 84.432} C_DIS
LIN {X -0.164,Y -414.873,Z 1712.455,A 0.000,B 0.000,C 90.000,E1 82.008} C_DIS
LIN {X 0.110,Y -395.667,Z 1712.439,A 0.000,B 0.000,C 90.000,E1 78.926} C_DIS
LIN {X -0.145,Y -380.832,Z 1712.424,A 0.000,B 0.000,C 90.000,E1 76.408} C_DIS
LIN {X -0.153,Y -366.523,Z 1712.410,A 0.000,B 0.000,C 90.000,E1 73.795} C_DIS
LIN {X -0.038,Y -354.157,Z 1712.397,A 0.000,B 0.000,C 90.000,E1 71.402} C_DIS
LIN {X 0.008,Y -339.342,Z 1712.380,A 0.000,B 0.000,C 90.000,E1 68.358} C_DIS
LIN {X 0.039,Y -327.830,Z 1712.366,A 0.000,B 0.000,C 90.000,E1 65.869} C_DIS
LIN {X 0.134,Y -315.338,Z 1712.350,A 0.000,B 0.000,C 90.000,E1 62.999} C_DIS
LIN {X -0.137,Y -304.433,Z 1712.336,A 0.000,B 0.000,C 90.000,E1 60.461} C_DIS
LIN {X 0.043,Y -293.618,Z 1712.321,A 0.000,B 0.000,C 90.000,E1 57.788} C_DIS
LIN {X -0.090,Y -285.393,Z 1712.310,A 0.000,B 0.000,C 90.000,E1 55.801} C_DIS
LIN {X -0.049,Y -277.036,Z 1712.299,A 0.000,B 0.000,C 90.000,E1 53.749} C_DIS
LIN {X -0.087,Y -267.165,Z 1712.285,A 0.000,B 0.000,C 90.000,E1 51.331} C_DIS
LIN {X -0.008,Y -255.996,Z 1712.269,A 0.000,B 0.000,C 90.000,E1 48.485} C_DIS
LIN {X 0.110,Y -245.233,Z 1712.253,A 0.000,B 0.000,C 90.000,E1 45.567} C_DIS
